LIN {X 35.400,Y 125.914,Z 53.000,A 180.000,B 0.000,C 180.000} C_DIS
LIN {X 35.221,Y 125.886,Z 53.000,A 180.000,B 0.000,C 180.000} C_DIS
LIN {X 35.056,Y 125.857,Z 53.000,A 180.000,B 0.000,C 180.000} C_DIS
LIN {X 34.685,Y 125.774,Z 53.000,A 180.000,B 0.000,C 180.000} C_DIS
LIN {X 34.506,Y 125.726,Z 53.000,A 180.000,B 0.000,C 180.000} C_DIS
LIN {X 34.327,Y 125.674,Z 53.000,A 180.000,B 0.000,C 180.000} C_DIS
LIN {X 34.148,Y 125.619,Z 53.000,A 180.000,B 0.000,C 180.000} C_DIS
LIN {X 33.791,Y 125.491,Z 53.000,A 180.000,B 0.000,C 180.000} C_DIS
LIN {X 33.612,Y 125.417,Z 53.000,A 180.000,B 0.000,C 180.000} C_DIS
LIN {X 33.390,Y 125.321,Z 53.000,A 180.000,B 0.000,C 180.000} C_DIS
LIN {X 33.254,Y 125.258,Z 53.000,A 180.000,B 0.000,C 180.000} C_DIS
LIN {X 32.897,Y 125.076,Z 53.000,A 180.000,B 0.000,C 180.000} C_DIS
LIN {X 32.718,Y 124.971,Z 53.000,A 180.000,B 0.000,C 180.000} C_DIS
LIN {X 32.539,Y 124.865,Z 53.000,A 180.000,B 0.000,C 180.000} C_DIS
LIN {X 32.413,Y 124.785,Z 53.000,A 180.000,B 0.000,C 180.000} C_DIS
LIN {X 32.150,Y 124.606,Z 53.000,A 180.000,B 0.000,C 180.000} C_DIS
LIN {X 32.003,Y 124.497,Z 53.000,A 180.000,B 0.000,C 180.000} C_DIS
LIN {X 31.824,Y 124.359,Z 53.000,A 180.000,B 0.000,C 180.000} C_DIS
LIN {X 31.687,Y 124.248,Z 53.000,A 180.000,B 0.000,C 180.000} C_DIS
LIN {X 31.467,Y 124.055,Z 53.000,A 180.000,B 0.000,C 180.000} C_DIS
LIN {X 31.291,Y 123.891,Z 53.000,A 180.000,B 0.000,C 180.000} C_DIS
LIN {X 31.109,Y 123.709,Z 53.000,A 180.000,B 0.000,C 180.000} C_DIS
LIN {X 30.945,Y 123.533,Z 53.000,A 180.000,B 0.000,C 180.000} C_DIS
LIN {X 30.752,Y 123.313,Z 53.000,A 180.000,B 0.000,C 180.000} C_DIS
LIN {X 30.641,Y 123.176,Z 53.000,A 180.000,B 0.000,C 180.000} C_DIS
LIN {X 30.503,Y 122.997,Z 53.000,A 180.000,B 0.000,C 180.000} C_DIS
LIN {X 30.394,Y 122.850,Z 53.000,A 180.000,B 0.000,C 180.000} C_DIS
LIN {X 30.215,Y 122.587,Z 53.000,A 180.000,B 0.000,C 180.000} C_DIS
LIN {X 30.135,Y 122.461,Z 53.000,A 180.000,B 0.000,C 180.000} C_DIS
LIN {X 30.029,Y 122.282,Z 53.000,A 180.000,B 0.000,C 180.000} C_DIS
LIN {X 29.924,Y 122.103,Z 53.000,A 180.000,B 0.000,C 180.000} C_DIS
LIN {X 29.742,Y 121.746,Z 53.000,A 180.000,B 0.000,C 180.000} C_DIS
LIN {X 29.679,Y 121.610,Z 53.000,A 180.000,B 0.000,C 180.000} C_DIS
LIN {X 29.583,Y 121.388,Z 53.000,A 180.000,B 0.000,C 180.000} C_DIS
LIN {X 29.509,Y 121.209,Z 53.000,A 180.000,B 0.000,C 180.000} C_DIS
LIN {X 29.381,Y 120.852,Z 53.000,A 180.000,B 0.000,C 180.000} C_DIS
LIN {X 29.326,Y 120.673,Z 53.000,A 180.000,B 0.000,C 180.000} C_DIS
LIN {X 29.274,Y 120.494,Z 53.000,A 180.000,B 0.000,C 180.000} C_DIS
LIN {X 29.226,Y 120.315,Z 53.000,A 180.000,B 0.000,C 180.000} C_DIS
LIN {X 29.143,Y 119.944,Z 53.000,A 180.000,B 0.000,C 180.000} C_DIS
LIN {X 29.114,Y 119.779,Z 53.000,A 180.000,B 0.000,C 180.000} C_DIS
LIN {X 29.086,Y 119.600,Z 53.000,A 180.000,B 0.000,C 180.000} C_DIS
LIN {X 29.059,Y 119.422,Z 53.000,A 180.000,B 0.000,C 180.000} C_DIS
LIN {X 29.025,Y 119.064,Z 53.000,A 180.000,B 0.000,C 180.000} C_DIS
LIN {X 29.013,Y 118.885,Z 53.000,A 180.000,B 0.000,C 180.000} C_DIS
LIN {X 29.002,Y 118.528,Z 53.000,A 180.000,B 0.000,C 180.000} C_DIS
LIN {X 29.006,Y 118.349,Z 53.000,A 180.000,B 0.000,C 180.000} C_DIS
LIN {X 29.012,Y 118.170,Z 53.000,A 180.000,B 0.000,C 180.000} C_DIS
LIN {X 29.020,Y 117.991,Z 53.000,A 180.000,B 0.000,C 180.000} C_DIS
LIN {X 29.053,Y 117.634,Z 53.000,A 180.000,B 0.000,C 180.000} C_DIS
LIN {X 29.077,Y 117.455,Z 53.000,A 180.000,B 0.000,C 180.000} C_DIS
LIN {X 29.134,Y 117.098,Z 53.000,A 180.000,B 0.000,C 180.000} C_DIS
LIN {X 29.143,Y 117.056,Z 53.000,A 180.000,B 0.000,C 180.000} C_DIS
LIN {X 29.213,Y 116.740,Z 53.000,A 180.000,B 0.000,C 180.000} C_DIS
LIN {X 29.258,Y 116.561,Z 53.000,A 180.000,B 0.000,C 180.000} C_DIS
LIN {X 29.362,Y 116.204,Z 53.000,A 180.000,B 0.000,C 180.000} C_DIS
LIN {X 29.425,Y 116.025,Z 53.000,A 180.000,B 0.000,C 180.000} C_DIS
LIN {X 29.500,Y 115.816,Z 53.000,A 180.000,B 0.000,C 180.000} C_DIS
LIN {X 29.559,Y 115.667,Z 53.000,A 180.000,B 0.000,C 180.000} C_DIS
LIN {X 29.714,Y 115.310,Z 53.000,A 180.000,B 0.000,C 180.000} C_DIS
LIN {X 29.805,Y 115.131,Z 53.000,A 180.000,B 0.000,C 180.000} C_DIS
LIN {X 29.896,Y 114.952,Z 53.000,A 180.000,B 0.000,C 180.000} C_DIS
LIN {X 29.996,Y 114.774,Z 53.000,A 180.000,B 0.000,C 180.000} C_DIS
LIN {X 30.102,Y 114.595,Z 53.000,A 180.000,B 0.000,C 180.000} C_DIS
LIN {X 30.213,Y 114.416,Z 53.000,A 180.000,B 0.000,C 180.000} C_DIS
LIN {X 30.394,Y 114.150,Z 53.000,A 180.000,B 0.000,C 180.000} C_DIS
LIN {X 30.460,Y 114.058,Z 53.000,A 180.000,B 0.000,C 180.000} C_DIS
LIN {X 30.598,Y 113.880,Z 53.000,A 180.000,B 0.000,C 180.000} C_DIS
LIN {X 30.739,Y 113.701,Z 53.000,A 180.000,B 0.000,C 180.000} C_DIS
LIN {X 30.930,Y 113.484,Z 53.000,A 180.000,B 0.000,C 180.000} C_DIS
LIN {X 31.057,Y 113.343,Z 53.000,A 180.000,B 0.000,C 180.000} C_DIS
LIN {X 31.288,Y 113.112,Z 53.000,A 180.000,B 0.000,C 180.000} C_DIS
LIN {X 31.421,Y 112.986,Z 53.000,A 180.000,B 0.000,C 180.000} C_DIS
LIN {X 31.646,Y 112.788,Z 53.000,A 180.000,B 0.000,C 180.000} C_DIS
LIN {X 31.824,Y 112.641,Z 53.000,A 180.000,B 0.000,C 180.000} C_DIS
LIN {X 32.072,Y 112.450,Z 53.000,A 180.000,B 0.000,C 180.000} C_DIS
LIN {X 32.182,Y 112.373,Z 53.000,A 180.000,B 0.000,C 180.000} C_DIS
LIN {X 32.361,Y 112.251,Z 53.000,A 180.000,B 0.000,C 180.000} C_DIS
LIN {X 32.539,Y 112.135,Z 53.000,A 180.000,B 0.000,C 180.000} C_DIS
LIN {X 32.718,Y 112.029,Z 53.000,A 180.000,B 0.000,C 180.000} C_DIS
LIN {X 32.897,Y 111.924,Z 53.000,A 180.000,B 0.000,C 180.000} C_DIS
LIN {X 33.269,Y 111.734,Z 53.000,A 180.000,B 0.000,C 180.000} C_DIS
LIN {X 33.433,Y 111.660,Z 53.000,A 180.000,B 0.000,C 180.000} C_DIS
LIN {X 33.675,Y 111.556,Z 53.000,A 180.000,B 0.000,C 180.000} C_DIS
LIN {X 33.791,Y 111.509,Z 53.000,A 180.000,B 0.000,C 180.000} C_DIS
LIN {X 34.159,Y 111.377,Z 53.000,A 180.000,B 0.000,C 180.000} C_DIS
LIN {X 34.327,Y 111.326,Z 53.000,A 180.000,B 0.000,C 180.000} C_DIS
LIN {X 34.506,Y 111.274,Z 53.000,A 180.000,B 0.000,C 180.000} C_DIS
LIN {X 34.685,Y 111.226,Z 53.000,A 180.000,B 0.000,C 180.000} C_DIS
LIN {X 35.042,Y 111.146,Z 53.000,A 180.000,B 0.000,C 180.000} C_DIS
LIN {X 35.221,Y 111.114,Z 53.000,A 180.000,B 0.000,C 180.000} C_DIS
LIN {X 35.400,Y 111.086,Z 53.000,A 180.000,B 0.000,C 180.000} C_DIS
LIN {X 35.578,Y 111.059,Z 53.000,A 180.000,B 0.000,C 180.000} C_DIS
LIN {X 35.994,Y 111.019,Z 53.000,A 180.000,B 0.000,C 180.000} C_DIS
LIN {X 36.115,Y 111.013,Z 53.000,A 180.000,B 0.000,C 180.000} C_DIS
LIN {X 36.472,Y 111.002,Z 53.000,A 180.000,B 0.000,C 180.000} C_DIS
LIN {X 36.651,Y 111.006,Z 53.000,A 180.000,B 0.000,C 180.000} C_DIS
LIN {X 36.830,Y 111.012,Z 53.000,A 180.000,B 0.000,C 180.000} C_DIS
LIN {X 37.006,Y 111.019,Z 53.000,A 180.000,B 0.000,C 180.000} C_DIS
LIN {X 37.366,Y 111.053,Z 53.000,A 180.000,B 0.000,C 180.000} C_DIS
LIN {X 37.545,Y 111.077,Z 53.000,A 180.000,B 0.000,C 180.000} C_DIS
LIN {X 37.902,Y 111.134,Z 53.000,A 180.000,B 0.000,C 180.000} C_DIS
LIN {X 38.081,Y 111.173,Z 53.000,A 180.000,B 0.000,C 180.000} C_DIS
LIN {X 38.260,Y 111.213,Z 53.000,A 180.000,B 0.000,C 180.000} C_DIS
LIN {X 38.439,Y 111.258,Z 53.000,A 180.000,B 0.000,C 180.000} C_DIS
LIN {X 38.796,Y 111.362,Z 53.000,A 180.000,B 0.000,C 180.000} C_DIS
LIN {X 38.841,Y 111.377,Z 53.000,A 180.000,B 0.000,C 180.000} C_DIS
LIN {X 39.154,Y 111.489,Z 53.000,A 180.000,B 0.000,C 180.000} C_DIS
LIN {X 39.325,Y 111.556,Z 53.000,A 180.000,B 0.000,C 180.000} C_DIS
LIN {X 39.690,Y 111.714,Z 53.000,A 180.000,B 0.000,C 180.000} C_DIS
LIN {X 39.731,Y 111.734,Z 53.000,A 180.000,B 0.000,C 180.000} C_DIS
LIN {X 40.082,Y 111.913,Z 53.000,A 180.000,B 0.000,C 180.000} C_DIS
LIN {X 40.226,Y 111.996,Z 53.000,A 180.000,B 0.000,C 180.000} C_DIS
LIN {X 40.405,Y 112.102,Z 53.000,A 180.000,B 0.000,C 180.000} C_DIS
LIN {X 40.584,Y 112.213,Z 53.000,A 180.000,B 0.000,C 180.000} C_DIS
LIN {X 40.763,Y 112.335,Z 53.000,A 180.000,B 0.000,C 180.000} C_DIS
LIN {X 40.928,Y 112.450,Z 53.000,A 180.000,B 0.000,C 180.000} C_DIS
LIN {X 41.159,Y 112.628,Z 53.000,A 180.000,B 0.000,C 180.000} C_DIS
LIN {X 41.299,Y 112.739,Z 53.000,A 180.000,B 0.000,C 180.000} C_DIS
LIN {X 41.579,Y 112.986,Z 53.000,A 180.000,B 0.000,C 180.000} C_DIS
LIN {X 41.657,Y 113.057,Z 53.000,A 180.000,B 0.000,C 180.000} C_DIS
LIN {X 41.943,Y 113.343,Z 53.000,A 180.000,B 0.000,C 180.000} C_DIS
LIN {X 42.014,Y 113.421,Z 53.000,A 180.000,B 0.000,C 180.000} C_DIS
LIN {X 42.261,Y 113.701,Z 53.000,A 180.000,B 0.000,C 180.000} C_DIS
LIN {X 42.372,Y 113.841,Z 53.000,A 180.000,B 0.000,C 180.000} C_DIS
LIN {X 42.550,Y 114.072,Z 53.000,A 180.000,B 0.000,C 180.000} C_DIS
LIN {X 42.665,Y 114.237,Z 53.000,A 180.000,B 0.000,C 180.000} C_DIS
LIN {X 42.787,Y 114.416,Z 53.000,A 180.000,B 0.000,C 180.000} C_DIS
LIN {X 42.898,Y 114.595,Z 53.000,A 180.000,B 0.000,C 180.000} C_DIS
LIN {X 43.004,Y 114.774,Z 53.000,A 180.000,B 0.000,C 180.000} C_DIS
LIN {X 43.087,Y 114.918,Z 53.000,A 180.000,B 0.000,C 180.000} C_DIS
LIN {X 43.266,Y 115.269,Z 53.000,A 180.000,B 0.000,C 180.000} C_DIS
LIN {X 43.286,Y 115.310,Z 53.000,A 180.000,B 0.000,C 180.000} C_DIS
LIN {X 43.444,Y 115.675,Z 53.000,A 180.000,B 0.000,C 180.000} C_DIS
LIN {X 43.511,Y 115.846,Z 53.000,A 180.000,B 0.000,C 180.000} C_DIS
LIN {X 43.623,Y 116.159,Z 53.000,A 180.000,B 0.000,C 180.000} C_DIS
LIN {X 43.638,Y 116.204,Z 53.000,A 180.000,B 0.000,C 180.000} C_DIS
LIN {X 43.742,Y 116.561,Z 53.000,A 180.000,B 0.000,C 180.000} C_DIS
LIN {X 43.787,Y 116.740,Z 53.000,A 180.000,B 0.000,C 180.000} C_DIS
LIN {X 43.827,Y 116.919,Z 53.000,A 180.000,B 0.000,C 180.000} C_DIS
LIN {X 43.866,Y 117.098,Z 53.000,A 180.000,B 0.000,C 180.000} C_DIS
LIN {X 43.923,Y 117.455,Z 53.000,A 180.000,B 0.000,C 180.000} C_DIS
LIN {X 43.947,Y 117.634,Z 53.000,A 180.000,B 0.000,C 180.000} C_DIS
LIN {X 43.981,Y 117.994,Z 53.000,A 180.000,B 0.000,C 180.000} C_DIS
LIN {X 43.988,Y 118.170,Z 53.000,A 180.000,B 0.000,C 180.000} C_DIS
LIN {X 43.994,Y 118.349,Z 53.000,A 180.000,B 0.000,C 180.000} C_DIS
LIN {X 43.998,Y 118.528,Z 53.000,A 180.000,B 0.000,C 180.000} C_DIS
LIN {X 43.987,Y 118.885,Z 53.000,A 180.000,B 0.000,C 180.000} C_DIS
LIN {X 43.981,Y 119.006,Z 53.000,A 180.000,B 0.000,C 180.000} C_DIS
LIN {X 43.941,Y 119.422,Z 53.000,A 180.000,B 0.000,C 180.000} C_DIS
LIN {X 43.914,Y 119.600,Z 53.000,A 180.000,B 0.000,C 180.000} C_DIS
LIN {X 43.886,Y 119.779,Z 53.000,A 180.000,B 0.000,C 180.000} C_DIS
LIN {X 43.854,Y 119.958,Z 53.000,A 180.000,B 0.000,C 180.000} C_DIS
LIN {X 43.774,Y 120.315,Z 53.000,A 180.000,B 0.000,C 180.000} C_DIS
LIN {X 43.726,Y 120.494,Z 53.000,A 180.000,B 0.000,C 180.000} C_DIS
LIN {X 43.674,Y 120.673,Z 53.000,A 180.000,B 0.000,C 180.000} C_DIS
LIN {X 43.623,Y 120.841,Z 53.000,A 180.000,B 0.000,C 180.000} C_DIS
LIN {X 43.491,Y 121.209,Z 53.000,A 180.000,B 0.000,C 180.000} C_DIS
LIN {X 43.444,Y 121.325,Z 53.000,A 180.000,B 0.000,C 180.000} C_DIS
LIN {X 43.340,Y 121.567,Z 53.000,A 180.000,B 0.000,C 180.000} C_DIS
LIN {X 43.266,Y 121.731,Z 53.000,A 180.000,B 0.000,C 180.000} C_DIS
LIN {X 43.076,Y 122.103,Z 53.000,A 180.000,B 0.000,C 180.000} C_DIS
LIN {X 42.971,Y 122.282,Z 53.000,A 180.000,B 0.000,C 180.000} C_DIS
LIN {X 42.865,Y 122.461,Z 53.000,A 180.000,B 0.000,C 180.000} C_DIS
LIN {X 42.749,Y 122.639,Z 53.000,A 180.000,B 0.000,C 180.000} C_DIS
LIN {X 42.627,Y 122.818,Z 53.000,A 180.000,B 0.000,C 180.000} C_DIS
LIN {X 42.550,Y 122.928,Z 53.000,A 180.000,B 0.000,C 180.000} C_DIS
LIN {X 42.359,Y 123.176,Z 53.000,A 180.000,B 0.000,C 180.000} C_DIS
LIN {X 42.212,Y 123.354,Z 53.000,A 180.000,B 0.000,C 180.000} C_DIS
LIN {X 42.014,Y 123.579,Z 53.000,A 180.000,B 0.000,C 180.000} C_DIS
LIN {X 41.888,Y 123.712,Z 53.000,A 180.000,B 0.000,C 180.000} C_DIS
LIN {X 41.870,Y 123.729,Z 53.000,A 180.000,B 0.000,C 180.000} C_DIS
; Link Move Starts
LIN {X 41.648,Y 123.952,Z 53.000,A 180.000,B 0.000,C 180.000} C_DIS
LIN {X 41.412,Y 124.161,Z 52.999,A 180.000,B 0.000,C 180.000} C_DIS
LIN {X 41.170,Y 124.363,Z 52.998,A 180.000,B 0.000,C 180.000} C_DIS
LIN {X 40.921,Y 124.556,Z 52.996,A 180.000,B 0.000,C 180.000} C_DIS
LIN {X 40.661,Y 124.734,Z 52.994,A 180.000,B 0.000,C 180.000} C_DIS
LIN {X 40.396,Y 124.904,Z 52.991,A 180.000,B 0.000,C 180.000} C_DIS
LIN {X 40.125,Y 125.064,Z 52.988,A 180.000,B 0.000,C 180.000} C_DIS
LIN {X 39.845,Y 125.208,Z 52.985,A 180.000,B 0.000,C 180.000} C_DIS
LIN {X 39.560,Y 125.343,Z 52.981,A 180.000,B 0.000,C 180.000} C_DIS
LIN {X 39.271,Y 125.468,Z 52.977,A 180.000,B 0.000,C 180.000} C_DIS
LIN {X 38.975,Y 125.575,Z 52.972,A 180.000,B 0.000,C 180.000} C_DIS
LIN {X 38.827,Y 125.628,Z 52.969,A 180.000,B 0.000,C 180.000} C_DIS
LIN {X 38.676,Y 125.673,Z 52.967,A 180.000,B 0.000,C 180.000} C_DIS
LIN {X 38.524,Y 125.717,Z 52.964,A 180.000,B 0.000,C 180.000} C_DIS
LIN {X 38.373,Y 125.761,Z 52.961,A 180.000,B 0.000,C 180.000} C_DIS
LIN {X 38.219,Y 125.796,Z 52.959,A 180.000,B 0.000,C 180.000} C_DIS
LIN {X 38.066,Y 125.830,Z 52.956,A 180.000,B 0.000,C 180.000} C_DIS
LIN {X 37.912,Y 125.864,Z 52.952,A 180.000,B 0.000,C 180.000} C_DIS
LIN {X 37.756,Y 125.889,Z 52.949,A 180.000,B 0.000,C 180.000} C_DIS
LIN {X 37.601,Y 125.914,Z 52.946,A 180.000,B 0.000,C 180.000} C_DIS
LIN {X 37.445,Y 125.939,Z 52.943,A 180.000,B 0.000,C 180.000} C_DIS
LIN {X 37.289,Y 125.954,Z 52.939,A 180.000,B 0.000,C 180.000} C_DIS
LIN {X 37.132,Y 125.969,Z 52.936,A 180.000,B 0.000,C 180.000} C_DIS
LIN {X 36.975,Y 125.984,Z 52.932,A 180.000,B 0.000,C 180.000} C_DIS
LIN {X 36.817,Y 125.989,Z 52.928,A 180.000,B 0.000,C 180.000} C_DIS
LIN {X 36.660,Y 125.994,Z 52.925,A 180.000,B 0.000,C 180.000} C_DIS
LIN {X 36.503,Y 125.999,Z 52.921,A 180.000,B 0.000,C 180.000} C_DIS
LIN {X 36.345,Y 125.994,Z 52.917,A 180.000,B 0.000,C 180.000} C_DIS
LIN {X 36.188,Y 125.989,Z 52.913,A 180.000,B 0.000,C 180.000} C_DIS
LIN {X 36.030,Y 125.984,Z 52.909,A 180.000,B 0.000,C 180.000} C_DIS
LIN {X 35.873,Y 125.969,Z 52.905,A 180.000,B 0.000,C 180.000} C_DIS
LIN {X 35.717,Y 125.954,Z 52.900,A 180.000,B 0.000,C 180.000} C_DIS
LIN {X 35.560,Y 125.940,Z 52.896,A 180.000,B 0.000,C 180.000} C_DIS
LIN {X 35.404,Y 125.915,Z 52.892,A 180.000,B 0.000,C 180.000} C_DIS
LIN {X 35.249,Y 125.890,Z 52.887,A 180.000,B 0.000,C 180.000} C_DIS
LIN {X 35.093,Y 125.866,Z 52.883,A 180.000,B 0.000,C 180.000} C_DIS
LIN {X 34.939,Y 125.831,Z 52.878,A 180.000,B 0.000,C 180.000} C_DIS
LIN {X 34.786,Y 125.797,Z 52.873,A 180.000,B 0.000,C 180.000} C_DIS
LIN {X 34.632,Y 125.762,Z 52.869,A 180.000,B 0.000,C 180.000} C_DIS
LIN {X 34.481,Y 125.718,Z 52.864,A 180.000,B 0.000,C 180.000} C_DIS
LIN {X 34.329,Y 125.674,Z 52.859,A 180.000,B 0.000,C 180.000} C_DIS
LIN {X 34.178,Y 125.630,Z 52.854,A 180.000,B 0.000,C 180.000} C_DIS
LIN {X 34.104,Y 125.603,Z 52.851,A 180.000,B 0.000,C 180.000} C_DIS
LIN {X 34.030,Y 125.577,Z 52.849,A 180.000,B 0.000,C 180.000} C_DIS
LIN {X 33.956,Y 125.550,Z 52.846,A 180.000,B 0.000,C 180.000} C_DIS
LIN {X 33.882,Y 125.523,Z 52.844,A 180.000,B 0.000,C 180.000} C_DIS
LIN {X 33.808,Y 125.497,Z 52.841,A 180.000,B 0.000,C 180.000} C_DIS
LIN {X 33.734,Y 125.470,Z 52.839,A 180.000,B 0.000,C 180.000} C_DIS
LIN {X 33.661,Y 125.438,Z 52.836,A 180.000,B 0.000,C 180.000} C_DIS
LIN {X 33.517,Y 125.376,Z 52.831,A 180.000,B 0.000,C 180.000} C_DIS
LIN {X 33.372,Y 125.313,Z 52.825,A 180.000,B 0.000,C 180.000} C_DIS
LIN {X 33.300,Y 125.282,Z 52.823,A 180.000,B 0.000,C 180.000} C_DIS
LIN {X 33.160,Y 125.210,Z 52.817,A 180.000,B 0.000,C 180.000} C_DIS
LIN {X 33.020,Y 125.139,Z 52.812,A 180.000,B 0.000,C 180.000} C_DIS
LIN {X 32.949,Y 125.103,Z 52.809,A 180.000,B 0.000,C 180.000} C_DIS
LIN {X 32.880,Y 125.067,Z 52.806,A 180.000,B 0.000,C 180.000} C_DIS
LIN {X 32.744,Y 124.986,Z 52.801,A 180.000,B 0.000,C 180.000} C_DIS
LIN {X 32.541,Y 124.866,Z 52.793,A 180.000,B 0.000,C 180.000} C_DIS
LIN {X 32.473,Y 124.825,Z 52.790,A 180.000,B 0.000,C 180.000} C_DIS
LIN {X 32.278,Y 124.693,Z 52.782,A 180.000,B 0.000,C 180.000} C_DIS
LIN {X 32.147,Y 124.604,Z 52.776,A 180.000,B 0.000,C 180.000} C_DIS
LIN {X 32.083,Y 124.559,Z 52.774,A 180.000,B 0.000,C 180.000} C_DIS
LIN {X 31.958,Y 124.463,Z 52.768,A 180.000,B 0.000,C 180.000} C_DIS
LIN {X 31.772,Y 124.318,Z 52.760,A 180.000,B 0.000,C 180.000} C_DIS
LIN {X 31.710,Y 124.269,Z 52.757,A 180.000,B 0.000,C 180.000} C_DIS
LIN {X 31.533,Y 124.113,Z 52.749,A 180.000,B 0.000,C 180.000} C_DIS
LIN {X 31.414,Y 124.008,Z 52.743,A 180.000,B 0.000,C 180.000} C_DIS
LIN {X 31.356,Y 123.956,Z 52.741,A 180.000,B 0.000,C 180.000} C_DIS
LIN {X 31.245,Y 123.844,Z 52.735,A 180.000,B 0.000,C 180.000} C_DIS
LIN {X 31.078,Y 123.677,Z 52.727,A 180.000,B 0.000,C 180.000} C_DIS
LIN {X 31.023,Y 123.621,Z 52.724,A 180.000,B 0.000,C 180.000} C_DIS
LIN {X 30.762,Y 123.325,Z 52.710,A 180.000,B 0.000,C 180.000} C_DIS
LIN {X 30.711,Y 123.265,Z 52.708,A 180.000,B 0.000,C 180.000} C_DIS
LIN {X 30.614,Y 123.141,Z 52.702,A 180.000,B 0.000,C 180.000} C_DIS
LIN {X 30.470,Y 122.954,Z 52.694,A 180.000,B 0.000,C 180.000} C_DIS
LIN {X 30.422,Y 122.891,Z 52.691,A 180.000,B 0.000,C 180.000} C_DIS
LIN {X 30.201,Y 122.566,Z 52.677,A 180.000,B 0.000,C 180.000} C_DIS
LIN {X 30.158,Y 122.500,Z 52.675,A 180.000,B 0.000,C 180.000} C_DIS
LIN {X 30.078,Y 122.364,Z 52.669,A 180.000,B 0.000,C 180.000} C_DIS
LIN {X 29.957,Y 122.161,Z 52.661,A 180.000,B 0.000,C 180.000} C_DIS
LIN {X 29.918,Y 122.092,Z 52.658,A 180.000,B 0.000,C 180.000} C_DIS
LIN {X 29.740,Y 121.742,Z 52.644,A 180.000,B 0.000,C 180.000} C_DIS
LIN {X 29.705,Y 121.671,Z 52.642,A 180.000,B 0.000,C 180.000} C_DIS
LIN {X 29.612,Y 121.454,Z 52.633,A 180.000,B 0.000,C 180.000} C_DIS
LIN {X 29.549,Y 121.309,Z 52.628,A 180.000,B 0.000,C 180.000} C_DIS
LIN {X 29.519,Y 121.236,Z 52.625,A 180.000,B 0.000,C 180.000} C_DIS
LIN {X 29.386,Y 120.866,Z 52.611,A 180.000,B 0.000,C 180.000} C_DIS
LIN {X 29.361,Y 120.791,Z 52.609,A 180.000,B 0.000,C 180.000} C_DIS
LIN {X 29.295,Y 120.564,Z 52.600,A 180.000,B 0.000,C 180.000} C_DIS
LIN {X 29.251,Y 120.413,Z 52.595,A 180.000,B 0.000,C 180.000} C_DIS
LIN {X 29.231,Y 120.337,Z 52.592,A 180.000,B 0.000,C 180.000} C_DIS
LIN {X 29.145,Y 119.953,Z 52.578,A 180.000,B 0.000,C 180.000} C_DIS
LIN {X 29.129,Y 119.875,Z 52.576,A 180.000,B 0.000,C 180.000} C_DIS
LIN {X 29.068,Y 119.487,Z 52.562,A 180.000,B 0.000,C 180.000} C_DIS
LIN {X 29.057,Y 119.408,Z 52.559,A 180.000,B 0.000,C 180.000} C_DIS
LIN {X 29.020,Y 119.016,Z 52.545,A 180.000,B 0.000,C 180.000} C_DIS
LIN {X 29.015,Y 118.938,Z 52.543,A 180.000,B 0.000,C 180.000} C_DIS
LIN {X 29.003,Y 118.544,Z 52.529,A 180.000,B 0.000,C 180.000} C_DIS
LIN {X 29.002,Y 118.466,Z 52.526,A 180.000,B 0.000,C 180.000} C_DIS
LIN {X 29.015,Y 118.072,Z 52.512,A 180.000,B 0.000,C 180.000} C_DIS
LIN {X 29.019,Y 117.993,Z 52.510,A 180.000,B 0.000,C 180.000} C_DIS
LIN {X 29.056,Y 117.601,Z 52.496,A 180.000,B 0.000,C 180.000} C_DIS
LIN {X 29.066,Y 117.523,Z 52.493,A 180.000,B 0.000,C 180.000} C_DIS
LIN {X 29.128,Y 117.134,Z 52.479,A 180.000,B 0.000,C 180.000} C_DIS
LIN {X 29.143,Y 117.057,Z 52.477,A 180.000,B 0.000,C 180.000} C_DIS
LIN {X 29.228,Y 116.673,Z 52.463,A 180.000,B 0.000,C 180.000} C_DIS
LIN {X 29.248,Y 116.596,Z 52.460,A 180.000,B 0.000,C 180.000} C_DIS
LIN {X 29.358,Y 116.218,Z 52.446,A 180.000,B 0.000,C 180.000} C_DIS
LIN {X 29.382,Y 116.143,Z 52.444,A 180.000,B 0.000,C 180.000} C_DIS
LIN {X 29.516,Y 115.773,Z 52.430,A 180.000,B 0.000,C 180.000} C_DIS
LIN {X 29.545,Y 115.700,Z 52.427,A 180.000,B 0.000,C 180.000} C_DIS
LIN {X 29.701,Y 115.338,Z 52.413,A 180.000,B 0.000,C 180.000} C_DIS
LIN {X 29.735,Y 115.267,Z 52.411,A 180.000,B 0.000,C 180.000} C_DIS
LIN {X 29.842,Y 115.057,Z 52.402,A 180.000,B 0.000,C 180.000} C_DIS
LIN {X 29.914,Y 114.916,Z 52.397,A 180.000,B 0.000,C 180.000} C_DIS
LIN {X 29.952,Y 114.848,Z 52.394,A 180.000,B 0.000,C 180.000} C_DIS
LIN {X 30.153,Y 114.509,Z 52.380,A 180.000,B 0.000,C 180.000} C_DIS
LIN {X 30.195,Y 114.442,Z 52.378,A 180.000,B 0.000,C 180.000} C_DIS
LIN {X 30.328,Y 114.247,Z 52.369,A 180.000,B 0.000,C 180.000} C_DIS
LIN {X 30.417,Y 114.117,Z 52.364,A 180.000,B 0.000,C 180.000} C_DIS
LIN {X 30.464,Y 114.053,Z 52.361,A 180.000,B 0.000,C 180.000} C_DIS
LIN {X 30.705,Y 113.742,Z 52.347,A 180.000,B 0.000,C 180.000} C_DIS
LIN {X 30.756,Y 113.682,Z 52.345,A 180.000,B 0.000,C 180.000} C_DIS
LIN {X 30.912,Y 113.505,Z 52.336,A 180.000,B 0.000,C 180.000} C_DIS
LIN {X 31.016,Y 113.387,Z 52.331,A 180.000,B 0.000,C 180.000} C_DIS
LIN {X 31.071,Y 113.330,Z 52.328,A 180.000,B 0.000,C 180.000} C_DIS
LIN {X 31.349,Y 113.051,Z 52.314,A 180.000,B 0.000,C 180.000} C_DIS
LIN {X 31.407,Y 112.998,Z 52.312,A 180.000,B 0.000,C 180.000} C_DIS
LIN {X 31.525,Y 112.894,Z 52.306,A 180.000,B 0.000,C 180.000} C_DIS
LIN {X 31.702,Y 112.738,Z 52.298,A 180.000,B 0.000,C 180.000} C_DIS
LIN {X 31.764,Y 112.688,Z 52.295,A 180.000,B 0.000,C 180.000} C_DIS
LIN {X 31.950,Y 112.543,Z 52.287,A 180.000,B 0.000,C 180.000} C_DIS
LIN {X 32.075,Y 112.447,Z 52.281,A 180.000,B 0.000,C 180.000} C_DIS
LIN {X 32.139,Y 112.402,Z 52.279,A 180.000,B 0.000,C 180.000} C_DIS
LIN {X 32.269,Y 112.313,Z 52.273,A 180.000,B 0.000,C 180.000} C_DIS
LIN {X 32.465,Y 112.180,Z 52.265,A 180.000,B 0.000,C 180.000} C_DIS
LIN {X 32.532,Y 112.139,Z 52.262,A 180.000,B 0.000,C 180.000} C_DIS
LIN {X 32.735,Y 112.019,Z 52.254,A 180.000,B 0.000,C 180.000} C_DIS
LIN {X 32.871,Y 111.939,Z 52.248,A 180.000,B 0.000,C 180.000} C_DIS
LIN {X 32.941,Y 111.902,Z 52.246,A 180.000,B 0.000,C 180.000} C_DIS
LIN {X 33.081,Y 111.830,Z 52.240,A 180.000,B 0.000,C 180.000} C_DIS
LIN {X 33.291,Y 111.723,Z 52.232,A 180.000,B 0.000,C 180.000} C_DIS
LIN {X 33.363,Y 111.691,Z 52.229,A 180.000,B 0.000,C 180.000} C_DIS
LIN {X 33.580,Y 111.597,Z 52.221,A 180.000,B 0.000,C 180.000} C_DIS
LIN {X 33.725,Y 111.534,Z 52.215,A 180.000,B 0.000,C 180.000} C_DIS
LIN {X 33.798,Y 111.507,Z 52.213,A 180.000,B 0.000,C 180.000} C_DIS
LIN {X 33.947,Y 111.453,Z 52.207,A 180.000,B 0.000,C 180.000} C_DIS
LIN {X 34.169,Y 111.373,Z 52.199,A 180.000,B 0.000,C 180.000} C_DIS
LIN {X 34.244,Y 111.350,Z 52.196,A 180.000,B 0.000,C 180.000} C_DIS
LIN {X 34.395,Y 111.306,Z 52.191,A 180.000,B 0.000,C 180.000} C_DIS
LIN {X 34.547,Y 111.263,Z 52.185,A 180.000,B 0.000,C 180.000} C_DIS
LIN {X 34.622,Y 111.241,Z 52.182,A 180.000,B 0.000,C 180.000} C_DIS
LIN {X 34.699,Y 111.223,Z 52.180,A 180.000,B 0.000,C 180.000} C_DIS
LIN {X 34.853,Y 111.188,Z 52.174,A 180.000,B 0.000,C 180.000} C_DIS
LIN {X 35.006,Y 111.154,Z 52.169,A 180.000,B 0.000,C 180.000} C_DIS
LIN {X 35.083,Y 111.137,Z 52.166,A 180.000,B 0.000,C 180.000} C_DIS
LIN {X 35.161,Y 111.124,Z 52.164,A 180.000,B 0.000,C 180.000} C_DIS
LIN {X 35.239,Y 111.111,Z 52.161,A 180.000,B 0.000,C 180.000} C_DIS
LIN {X 35.317,Y 111.099,Z 52.159,A 180.000,B 0.000,C 180.000} C_DIS
LIN {X 35.394,Y 111.087,Z 52.156,A 180.000,B 0.000,C 180.000} C_DIS
LIN {X 35.472,Y 111.074,Z 52.154,A 180.000,B 0.000,C 180.000} C_DIS
LIN {X 35.550,Y 111.062,Z 52.151,A 180.000,B 0.000,C 180.000} C_DIS
LIN {X 35.628,Y 111.054,Z 52.149,A 180.000,B 0.000,C 180.000} C_DIS
LIN {X 35.785,Y 111.039,Z 52.144,A 180.000,B 0.000,C 180.000} C_DIS
LIN {X 35.942,Y 111.024,Z 52.139,A 180.000,B 0.000,C 180.000} C_DIS
LIN {X 36.099,Y 111.014,Z 52.134,A 180.000,B 0.000,C 180.000} C_DIS
LIN {X 36.256,Y 111.009,Z 52.129,A 180.000,B 0.000,C 180.000} C_DIS
LIN {X 36.414,Y 111.004,Z 52.124,A 180.000,B 0.000,C 180.000} C_DIS
LIN {X 36.571,Y 111.003,Z 52.120,A 180.000,B 0.000,C 180.000} C_DIS
LIN {X 36.729,Y 111.008,Z 52.115,A 180.000,B 0.000,C 180.000} C_DIS
LIN {X 36.886,Y 111.013,Z 52.111,A 180.000,B 0.000,C 180.000} C_DIS
LIN {X 37.043,Y 111.023,Z 52.106,A 180.000,B 0.000,C 180.000} C_DIS
LIN {X 37.200,Y 111.038,Z 52.102,A 180.000,B 0.000,C 180.000} C_DIS
LIN {X 37.357,Y 111.053,Z 52.097,A 180.000,B 0.000,C 180.000} C_DIS
LIN {X 37.513,Y 111.072,Z 52.093,A 180.000,B 0.000,C 180.000} C_DIS
LIN {X 37.669,Y 111.097,Z 52.089,A 180.000,B 0.000,C 180.000} C_DIS
LIN {X 37.824,Y 111.121,Z 52.085,A 180.000,B 0.000,C 180.000} C_DIS
LIN {X 37.979,Y 111.151,Z 52.081,A 180.000,B 0.000,C 180.000} C_DIS
LIN {X 38.133,Y 111.185,Z 52.077,A 180.000,B 0.000,C 180.000} C_DIS
LIN {X 38.286,Y 111.219,Z 52.073,A 180.000,B 0.000,C 180.000} C_DIS
LIN {X 38.439,Y 111.258,Z 52.070,A 180.000,B 0.000,C 180.000} C_DIS
LIN {X 38.590,Y 111.302,Z 52.066,A 180.000,B 0.000,C 180.000} C_DIS
LIN {X 38.742,Y 111.346,Z 52.062,A 180.000,B 0.000,C 180.000} C_DIS
LIN {X 38.891,Y 111.395,Z 52.059,A 180.000,B 0.000,C 180.000} C_DIS
LIN {X 39.039,Y 111.448,Z 52.056,A 180.000,B 0.000,C 180.000} C_DIS
LIN {X 39.188,Y 111.502,Z 52.052,A 180.000,B 0.000,C 180.000} C_DIS
LIN {X 39.334,Y 111.560,Z 52.049,A 180.000,B 0.000,C 180.000} C_DIS
LIN {X 39.479,Y 111.622,Z 52.046,A 180.000,B 0.000,C 180.000} C_DIS
LIN {X 39.623,Y 111.685,Z 52.043,A 180.000,B 0.000,C 180.000} C_DIS
LIN {X 39.766,Y 111.752,Z 52.040,A 180.000,B 0.000,C 180.000} C_DIS
LIN {X 39.906,Y 111.823,Z 52.037,A 180.000,B 0.000,C 180.000} C_DIS
LIN {X 40.046,Y 111.895,Z 52.034,A 180.000,B 0.000,C 180.000} C_DIS
LIN {X 40.184,Y 111.971,Z 52.032,A 180.000,B 0.000,C 180.000} C_DIS
LIN {X 40.320,Y 112.051,Z 52.029,A 180.000,B 0.000,C 180.000} C_DIS
LIN {X 40.455,Y 112.131,Z 52.027,A 180.000,B 0.000,C 180.000} C_DIS
LIN {X 40.718,Y 112.305,Z 52.022,A 180.000,B 0.000,C 180.000} C_DIS
LIN {X 40.976,Y 112.486,Z 52.018,A 180.000,B 0.000,C 180.000} C_DIS
LIN {X 41.225,Y 112.679,Z 52.014,A 180.000,B 0.000,C 180.000} C_DIS
LIN {X 41.464,Y 112.884,Z 52.011,A 180.000,B 0.000,C 180.000} C_DIS
LIN {X 41.696,Y 113.097,Z 52.008,A 180.000,B 0.000,C 180.000} C_DIS
LIN {X 41.919,Y 113.319,Z 52.005,A 180.000,B 0.000,C 180.000} C_DIS
LIN {X 42.130,Y 113.553,Z 52.003,A 180.000,B 0.000,C 180.000} C_DIS
LIN {X 42.334,Y 113.793,Z 52.002,A 180.000,B 0.000,C 180.000} C_DIS
LIN {X 42.527,Y 114.042,Z 52.001,A 180.000,B 0.000,C 180.000} C_DIS
LIN {X 42.708,Y 114.300,Z 52.000,A 180.000,B 0.000,C 180.000} C_DIS
LIN {X 42.835,Y 114.494,Z 52.000,A 180.000,B 0.000,C 180.000} C_DIS
; Cutting Move Starts
LIN {X 42.898,Y 114.595,Z 52.000,A 180.000,B 0.000,C 180.000} C_DIS
LIN {X 43.004,Y 114.774,Z 52.000,A 180.000,B 0.000,C 180.000} C_DIS
LIN {X 43.087,Y 114.918,Z 52.000,A 180.000,B 0.000,C 180.000} C_DIS
LIN {X 43.266,Y 115.269,Z 52.000,A 180.000,B 0.000,C 180.000} C_DIS
LIN {X 43.286,Y 115.310,Z 52.000,A 180.000,B 0.000,C 180.000} C_DIS
LIN {X 43.444,Y 115.675,Z 52.000,A 180.000,B 0.000,C 180.000} C_DIS
LIN {X 43.511,Y 115.846,Z 52.000,A 180.000,B 0.000,C 180.000} C_DIS
LIN {X 43.623,Y 116.159,Z 52.000,A 180.000,B 0.000,C 180.000} C_DIS
LIN {X 43.638,Y 116.204,Z 52.000,A 180.000,B 0.000,C 180.000} C_DIS
LIN {X 43.742,Y 116.561,Z 52.000,A 180.000,B 0.000,C 180.000} C_DIS
LIN {X 43.787,Y 116.740,Z 52.000,A 180.000,B 0.000,C 180.000} C_DIS
LIN {X 43.827,Y 116.919,Z 52.000,A 180.000,B 0.000,C 180.000} C_DIS
LIN {X 43.866,Y 117.098,Z 52.000,A 180.000,B 0.000,C 180.000} C_DIS
LIN {X 43.923,Y 117.455,Z 52.000,A 180.000,B 0.000,C 180.000} C_DIS
LIN {X 43.947,Y 117.634,Z 52.000,A 180.000,B 0.000,C 180.000} C_DIS
LIN {X 43.981,Y 117.994,Z 52.000,A 180.000,B 0.000,C 180.000} C_DIS
LIN {X 43.988,Y 118.170,Z 52.000,A 180.000,B 0.000,C 180.000} C_DIS
LIN {X 43.994,Y 118.349,Z 52.000,A 180.000,B 0.000,C 180.000} C_DIS
LIN {X 43.998,Y 118.528,Z 52.000,A 180.000,B 0.000,C 180.000} C_DIS
LIN {X 43.987,Y 118.885,Z 52.000,A 180.000,B 0.000,C 180.000} C_DIS
LIN {X 43.981,Y 119.006,Z 52.000,A 180.000,B 0.000,C 180.000} C_DIS
LIN {X 43.941,Y 119.422,Z 52.000,A 180.000,B 0.000,C 180.000} C_DIS
LIN {X 43.914,Y 119.600,Z 52.000,A 180.000,B 0.000,C 180.000} C_DIS
LIN {X 43.886,Y 119.779,Z 52.000,A 180.000,B 0.000,C 180.000} C_DIS
LIN {X 43.854,Y 119.958,Z 52.000,A 180.000,B 0.000,C 180.000} C_DIS
LIN {X 43.774,Y 120.315,Z 52.000,A 180.000,B 0.000,C 180.000} C_DIS
LIN {X 43.726,Y 120.494,Z 52.000,A 180.000,B 0.000,C 180.000} C_DIS
LIN {X 43.674,Y 120.673,Z 52.000,A 180.000,B 0.000,C 180.000} C_DIS
LIN {X 43.623,Y 120.841,Z 52.000,A 180.000,B 0.000,C 180.000} C_DIS
LIN {X 43.491,Y 121.209,Z 52.000,A 180.000,B 0.000,C 180.000} C_DIS
LIN {X 43.444,Y 121.325,Z 52.000,A 180.000,B 0.000,C 180.000} C_DIS
LIN {X 43.340,Y 121.567,Z 52.000,A 180.000,B 0.000,C 180.000} C_DIS
LIN {X 43.266,Y 121.731,Z 52.000,A 180.000,B 0.000,C 180.000} C_DIS
LIN {X 43.076,Y 122.103,Z 52.000,A 180.000,B 0.000,C 180.000} C_DIS
LIN {X 42.971,Y 122.282,Z 52.000,A 180.000,B 0.000,C 180.000} C_DIS
LIN {X 42.865,Y 122.461,Z 52.000,A 180.000,B 0.000,C 180.000} C_DIS
LIN {X 42.749,Y 122.639,Z 52.000,A 180.000,B 0.000,C 180.000} C_DIS
LIN {X 42.627,Y 122.818,Z 52.000,A 180.000,B 0.000,C 180.000} C_DIS
LIN {X 42.550,Y 122.928,Z 52.000,A 180.000,B 0.000,C 180.000} C_DIS
LIN {X 42.359,Y 123.176,Z 52.000,A 180.000,B 0.000,C 180.000} C_DIS
LIN {X 42.212,Y 123.354,Z 52.000,A 180.000,B 0.000,C 180.000} C_DIS
LIN {X 42.014,Y 123.579,Z 52.000,A 180.000,B 0.000,C 180.000} C_DIS
LIN {X 41.888,Y 123.712,Z 52.000,A 180.000,B 0.000,C 180.000} C_DIS
LIN {X 41.657,Y 123.943,Z 52.000,A 180.000,B 0.000,C 180.000} C_DIS
LIN {X 41.516,Y 124.070,Z 52.000,A 180.000,B 0.000,C 180.000} C_DIS
LIN {X 41.299,Y 124.261,Z 52.000,A 180.000,B 0.000,C 180.000} C_DIS
LIN {X 41.120,Y 124.402,Z 52.000,A 180.000,B 0.000,C 180.000} C_DIS
LIN {X 40.942,Y 124.540,Z 52.000,A 180.000,B 0.000,C 180.000} C_DIS
LIN {X 40.850,Y 124.606,Z 52.000,A 180.000,B 0.000,C 180.000} C_DIS
LIN {X 40.584,Y 124.787,Z 52.000,A 180.000,B 0.000,C 180.000} C_DIS
LIN {X 40.405,Y 124.898,Z 52.000,A 180.000,B 0.000,C 180.000} C_DIS
LIN {X 40.226,Y 125.004,Z 52.000,A 180.000,B 0.000,C 180.000} C_DIS
LIN {X 40.048,Y 125.104,Z 52.000,A 180.000,B 0.000,C 180.000} C_DIS
LIN {X 39.869,Y 125.195,Z 52.000,A 180.000,B 0.000,C 180.000} C_DIS
LIN {X 39.690,Y 125.286,Z 52.000,A 180.000,B 0.000,C 180.000} C_DIS
LIN {X 39.333,Y 125.441,Z 52.000,A 180.000,B 0.000,C 180.000} C_DIS
LIN {X 39.184,Y 125.500,Z 52.000,A 180.000,B 0.000,C 180.000} C_DIS
LIN {X 38.975,Y 125.575,Z 52.000,A 180.000,B 0.000,C 180.000} C_DIS
LIN {X 38.796,Y 125.638,Z 52.000,A 180.000,B 0.000,C 180.000} C_DIS
LIN {X 38.439,Y 125.742,Z 52.000,A 180.000,B 0.000,C 180.000} C_DIS
LIN {X 38.260,Y 125.787,Z 52.000,A 180.000,B 0.000,C 180.000} C_DIS
LIN {X 37.944,Y 125.857,Z 52.000,A 180.000,B 0.000,C 180.000} C_DIS
LIN {X 37.902,Y 125.866,Z 52.000,A 180.000,B 0.000,C 180.000} C_DIS
LIN {X 37.545,Y 125.923,Z 52.000,A 180.000,B 0.000,C 180.000} C_DIS
LIN {X 37.366,Y 125.947,Z 52.000,A 180.000,B 0.000,C 180.000} C_DIS
LIN {X 37.009,Y 125.980,Z 52.000,A 180.000,B 0.000,C 180.000} C_DIS
LIN {X 36.830,Y 125.988,Z 52.000,A 180.000,B 0.000,C 180.000} C_DIS
LIN {X 36.651,Y 125.994,Z 52.000,A 180.000,B 0.000,C 180.000} C_DIS
LIN {X 36.472,Y 125.998,Z 52.000,A 180.000,B 0.000,C 180.000} C_DIS
LIN {X 36.115,Y 125.987,Z 52.000,A 180.000,B 0.000,C 180.000} C_DIS
LIN {X 35.936,Y 125.975,Z 52.000,A 180.000,B 0.000,C 180.000} C_DIS
LIN {X 35.578,Y 125.941,Z 52.000,A 180.000,B 0.000,C 180.000} C_DIS
LIN {X 35.400,Y 125.914,Z 52.000,A 180.000,B 0.000,C 180.000} C_DIS
LIN {X 35.221,Y 125.886,Z 52.000,A 180.000,B 0.000,C 180.000} C_DIS
LIN {X 35.056,Y 125.857,Z 52.000,A 180.000,B 0.000,C 180.000} C_DIS
LIN {X 34.685,Y 125.774,Z 52.000,A 180.000,B 0.000,C 180.000} C_DIS
LIN {X 34.506,Y 125.726,Z 52.000,A 180.000,B 0.000,C 180.000} C_DIS
LIN {X 34.327,Y 125.674,Z 52.000,A 180.000,B 0.000,C 180.000} C_DIS
LIN {X 34.148,Y 125.619,Z 52.000,A 180.000,B 0.000,C 180.000} C_DIS
LIN {X 33.791,Y 125.491,Z 52.000,A 180.000,B 0.000,C 180.000} C_DIS
LIN {X 33.612,Y 125.417,Z 52.000,A 180.000,B 0.000,C 180.000} C_DIS
LIN {X 33.390,Y 125.321,Z 52.000,A 180.000,B 0.000,C 180.000} C_DIS
LIN {X 33.254,Y 125.258,Z 52.000,A 180.000,B 0.000,C 180.000} C_DIS
LIN {X 32.897,Y 125.076,Z 52.000,A 180.000,B 0.000,C 180.000} C_DIS
LIN {X 32.718,Y 124.971,Z 52.000,A 180.000,B 0.000,C 180.000} C_DIS
LIN {X 32.539,Y 124.865,Z 52.000,A 180.000,B 0.000,C 180.000} C_DIS
LIN {X 32.413,Y 124.785,Z 52.000,A 180.000,B 0.000,C 180.000} C_DIS
LIN {X 32.150,Y 124.606,Z 52.000,A 180.000,B 0.000,C 180.000} C_DIS
LIN {X 32.003,Y 124.497,Z 52.000,A 180.000,B 0.000,C 180.000} C_DIS
LIN {X 31.824,Y 124.359,Z 52.000,A 180.000,B 0.000,C 180.000} C_DIS
LIN {X 31.687,Y 124.248,Z 52.000,A 180.000,B 0.000,C 180.000} C_DIS
LIN {X 31.467,Y 124.055,Z 52.000,A 180.000,B 0.000,C 180.000} C_DIS
LIN {X 31.291,Y 123.891,Z 52.000,A 180.000,B 0.000,C 180.000} C_DIS
LIN {X 31.109,Y 123.709,Z 52.000,A 180.000,B 0.000,C 180.000} C_DIS
LIN {X 30.945,Y 123.533,Z 52.000,A 180.000,B 0.000,C 180.000} C_DIS
LIN {X 30.752,Y 123.313,Z 52.000,A 180.000,B 0.000,C 180.000} C_DIS
LIN {X 30.641,Y 123.176,Z 52.000,A 180.000,B 0.000,C 180.000} C_DIS
LIN {X 30.503,Y 122.997,Z 52.000,A 180.000,B 0.000,C 180.000} C_DIS
LIN {X 30.394,Y 122.850,Z 52.000,A 180.000,B 0.000,C 180.000} C_DIS
LIN {X 30.215,Y 122.587,Z 52.000,A 180.000,B 0.000,C 180.000} C_DIS
LIN {X 30.135,Y 122.461,Z 52.000,A 180.000,B 0.000,C 180.000} C_DIS
LIN {X 30.029,Y 122.282,Z 52.000,A 180.000,B 0.000,C 180.000} C_DIS
LIN {X 29.924,Y 122.103,Z 52.000,A 180.000,B 0.000,C 180.000} C_DIS
LIN {X 29.742,Y 121.746,Z 52.000,A 180.000,B 0.000,C 180.000} C_DIS
LIN {X 29.679,Y 121.610,Z 52.000,A 180.000,B 0.000,C 180.000} C_DIS
LIN {X 29.583,Y 121.388,Z 52.000,A 180.000,B 0.000,C 180.000} C_DIS
LIN {X 29.509,Y 121.209,Z 52.000,A 180.000,B 0.000,C 180.000} C_DIS
LIN {X 29.381,Y 120.852,Z 52.000,A 180.000,B 0.000,C 180.000} C_DIS
LIN {X 29.326,Y 120.673,Z 52.000,A 180.000,B 0.000,C 180.000} C_DIS
LIN {X 29.274,Y 120.494,Z 52.000,A 180.000,B 0.000,C 180.000} C_DIS
LIN {X 29.226,Y 120.315,Z 52.000,A 180.000,B 0.000,C 180.000} C_DIS
LIN {X 29.143,Y 119.944,Z 52.000,A 180.000,B 0.000,C 180.000} C_DIS
LIN {X 29.114,Y 119.779,Z 52.000,A 180.000,B 0.000,C 180.000} C_DIS
LIN {X 29.086,Y 119.600,Z 52.000,A 180.000,B 0.000,C 180.000} C_DIS
LIN {X 29.059,Y 119.422,Z 52.000,A 180.000,B 0.000,C 180.000} C_DIS
LIN {X 29.025,Y 119.064,Z 52.000,A 180.000,B 0.000,C 180.000} C_DIS
LIN {X 29.013,Y 118.885,Z 52.000,A 180.000,B 0.000,C 180.000} C_DIS
LIN {X 29.002,Y 118.528,Z 52.000,A 180.000,B 0.000,C 180.000} C_DIS
LIN {X 29.006,Y 118.349,Z 52.000,A 180.000,B 0.000,C 180.000} C_DIS
LIN {X 29.012,Y 118.170,Z 52.000,A 180.000,B 0.000,C 180.000} C_DIS
LIN {X 29.020,Y 117.991,Z 52.000,A 180.000,B 0.000,C 180.000} C_DIS
LIN {X 29.053,Y 117.634,Z 52.000,A 180.000,B 0.000,C 180.000} C_DIS
LIN {X 29.077,Y 117.455,Z 52.000,A 180.000,B 0.000,C 180.000} C_DIS
LIN {X 29.134,Y 117.098,Z 52.000,A 180.000,B 0.000,C 180.000} C_DIS
LIN {X 29.143,Y 117.056,Z 52.000,A 180.000,B 0.000,C 180.000} C_DIS
LIN {X 29.213,Y 116.740,Z 52.000,A 180.000,B 0.000,C 180.000} C_DIS
LIN {X 29.258,Y 116.561,Z 52.000,A 180.000,B 0.000,C 180.000} C_DIS
LIN {X 29.362,Y 116.204,Z 52.000,A 180.000,B 0.000,C 180.000} C_DIS
LIN {X 29.425,Y 116.025,Z 52.000,A 180.000,B 0.000,C 180.000} C_DIS
LIN {X 29.500,Y 115.816,Z 52.000,A 180.000,B 0.000,C 180.000} C_DIS
LIN {X 29.559,Y 115.667,Z 52.000,A 180.000,B 0.000,C 180.000} C_DIS
LIN {X 29.714,Y 115.310,Z 52.000,A 180.000,B 0.000,C 180.000} C_DIS
LIN {X 29.805,Y 115.131,Z 52.000,A 180.000,B 0.000,C 180.000} C_DIS
LIN {X 29.896,Y 114.952,Z 52.000,A 180.000,B 0.000,C 180.000} C_DIS
LIN {X 29.996,Y 114.774,Z 52.000,A 180.000,B 0.000,C 180.000} C_DIS
LIN {X 30.102,Y 114.595,Z 52.000,A 180.000,B 0.000,C 180.000} C_DIS
LIN {X 30.213,Y 114.416,Z 52.000,A 180.000,B 0.000,C 180.000} C_DIS
LIN {X 30.394,Y 114.150,Z 52.000,A 180.000,B 0.000,C 180.000} C_DIS
LIN {X 30.460,Y 114.058,Z 52.000,A 180.000,B 0.000,C 180.000} C_DIS
LIN {X 30.598,Y 113.880,Z 52.000,A 180.000,B 0.000,C 180.000} C_DIS
LIN {X 30.739,Y 113.701,Z 52.000,A 180.000,B 0.000,C 180.000} C_DIS
LIN {X 30.930,Y 113.484,Z 52.000,A 180.000,B 0.000,C 180.000} C_DIS
LIN {X 31.057,Y 113.343,Z 52.000,A 180.000,B 0.000,C 180.000} C_DIS
LIN {X 31.288,Y 113.112,Z 52.000,A 180.000,B 0.000,C 180.000} C_DIS
LIN {X 31.421,Y 112.986,Z 52.000,A 180.000,B 0.000,C 180.000} C_DIS
LIN {X 31.646,Y 112.788,Z 52.000,A 180.000,B 0.000,C 180.000} C_DIS
LIN {X 31.824,Y 112.641,Z 52.000,A 180.000,B 0.000,C 180.000} C_DIS
LIN {X 32.072,Y 112.450,Z 52.000,A 180.000,B 0.000,C 180.000} C_DIS
LIN {X 32.182,Y 112.373,Z 52.000,A 180.000,B 0.000,C 180.000} C_DIS
LIN {X 32.361,Y 112.251,Z 52.000,A 180.000,B 0.000,C 180.000} C_DIS
LIN {X 32.539,Y 112.135,Z 52.000,A 180.000,B 0.000,C 180.000} C_DIS
LIN {X 32.718,Y 112.029,Z 52.000,A 180.000,B 0.000,C 180.000} C_DIS
LIN {X 32.897,Y 111.924,Z 52.000,A 180.000,B 0.000,C 180.000} C_DIS
LIN {X 33.269,Y 111.734,Z 52.000,A 180.000,B 0.000,C 180.000} C_DIS
LIN {X 33.433,Y 111.660,Z 52.000,A 180.000,B 0.000,C 180.000} C_DIS
LIN {X 33.675,Y 111.556,Z 52.000,A 180.000,B 0.000,C 180.000} C_DIS
LIN {X 33.791,Y 111.509,Z 52.000,A 180.000,B 0.000,C 180.000} C_DIS
LIN {X 34.159,Y 111.377,Z 52.000,A 180.000,B 0.000,C 180.000} C_DIS
LIN {X 34.327,Y 111.326,Z 52.000,A 180.000,B 0.000,C 180.000} C_DIS
LIN {X 34.506,Y 111.274,Z 52.000,A 180.000,B 0.000,C 180.000} C_DIS
LIN {X 34.685,Y 111.226,Z 52.000,A 180.000,B 0.000,C 180.000} C_DIS
LIN {X 35.042,Y 111.146,Z 52.000,A 180.000,B 0.000,C 180.000} C_DIS
LIN {X 35.221,Y 111.114,Z 52.000,A 180.000,B 0.000,C 180.000} C_DIS
LIN {X 35.400,Y 111.086,Z 52.000,A 180.000,B 0.000,C 180.000} C_DIS
LIN {X 35.578,Y 111.059,Z 52.000,A 180.000,B 0.000,C 180.000} C_DIS
LIN {X 35.994,Y 111.019,Z 52.000,A 180.000,B 0.000,C 180.000} C_DIS
LIN {X 36.115,Y 111.013,Z 52.000,A 180.000,B 0.000,C 180.000} C_DIS
LIN {X 36.472,Y 111.002,Z 52.000,A 180.000,B 0.000,C 180.000} C_DIS
LIN {X 36.651,Y 111.006,Z 52.000,A 180.000,B 0.000,C 180.000} C_DIS
LIN {X 36.830,Y 111.012,Z 52.000,A 180.000,B 0.000,C 180.000} C_DIS
LIN {X 37.006,Y 111.019,Z 52.000,A 180.000,B 0.000,C 180.000} C_DIS
LIN {X 37.366,Y 111.053,Z 52.000,A 180.000,B 0.000,C 180.000} C_DIS
LIN {X 37.545,Y 111.077,Z 52.000,A 180.000,B 0.000,C 180.000} C_DIS
LIN {X 37.902,Y 111.134,Z 52.000,A 180.000,B 0.000,C 180.000} C_DIS
LIN {X 38.081,Y 111.173,Z 52.000,A 180.000,B 0.000,C 180.000} C_DIS
LIN {X 38.260,Y 111.213,Z 52.000,A 180.000,B 0.000,C 180.000} C_DIS
LIN {X 38.439,Y 111.258,Z 52.000,A 180.000,B 0.000,C 180.000} C_DIS
LIN {X 38.796,Y 111.362,Z 52.000,A 180.000,B 0.000,C 180.000} C_DIS
LIN {X 38.841,Y 111.377,Z 52.000,A 180.000,B 0.000,C 180.000} C_DIS
LIN {X 39.154,Y 111.489,Z 52.000,A 180.000,B 0.000,C 180.000} C_DIS
LIN {X 39.325,Y 111.556,Z 52.000,A 180.000,B 0.000,C 180.000} C_DIS
LIN {X 39.690,Y 111.714,Z 52.000,A 180.000,B 0.000,C 180.000} C_DIS
LIN {X 39.731,Y 111.734,Z 52.000,A 180.000,B 0.000,C 180.000} C_DIS
LIN {X 40.082,Y 111.913,Z 52.000,A 180.000,B 0.000,C 180.000} C_DIS
LIN {X 40.226,Y 111.996,Z 52.000,A 180.000,B 0.000,C 180.000} C_DIS
LIN {X 40.405,Y 112.102,Z 52.000,A 180.000,B 0.000,C 180.000} C_DIS
LIN {X 40.584,Y 112.213,Z 52.000,A 180.000,B 0.000,C 180.000} C_DIS
LIN {X 40.763,Y 112.335,Z 52.000,A 180.000,B 0.000,C 180.000} C_DIS
LIN {X 40.928,Y 112.450,Z 52.000,A 180.000,B 0.000,C 180.000} C_DIS
LIN {X 41.159,Y 112.628,Z 52.000,A 180.000,B 0.000,C 180.000} C_DIS
LIN {X 41.299,Y 112.739,Z 52.000,A 180.000,B 0.000,C 180.000} C_DIS
LIN {X 41.579,Y 112.986,Z 52.000,A 180.000,B 0.000,C 180.000} C_DIS
LIN {X 41.657,Y 113.057,Z 52.000,A 180.000,B 0.000,C 180.000} C_DIS
LIN {X 41.943,Y 113.343,Z 52.000,A 180.000,B 0.000,C 180.000} C_DIS
LIN {X 42.014,Y 113.421,Z 52.000,A 180.000,B 0.000,C 180.000} C_DIS
LIN {X 42.261,Y 113.701,Z 52.000,A 180.000,B 0.000,C 180.000} C_DIS
LIN {X 42.372,Y 113.841,Z 52.000,A 180.000,B 0.000,C 180.000} C_DIS
LIN {X 42.550,Y 114.072,Z 52.000,A 180.000,B 0.000,C 180.000} C_DIS
LIN {X 42.665,Y 114.237,Z 52.000,A 180.000,B 0.000,C 180.000} C_DIS
LIN {X 42.787,Y 114.416,Z 52.000,A 180.000,B 0.000,C 180.000} C_DIS
LIN {X 42.835,Y 114.494,Z 52.000,A 180.000,B 0.000,C 180.000} C_DIS
; Lead Out Move Starts
LIN {X 42.872,Y 114.952,Z 52.000,A 180.000,B 0.000,C 180.000} C_DIS
LIN {X 42.519,Y 115.247,Z 52.000,A 180.000,B 0.000,C 180.000} C_DIS
LIN {X 41.626,Y 115.444,Z 52.000,A 180.000,B 0.000,C 180.000} C_DIS
LIN {X 41.281,Y 115.521,Z 52.146,A 180.000,B 0.000,C 180.000} C_DIS
LIN {X 41.138,Y 115.552,Z 52.500,A 180.000,B 0.000,C 180.000} C_DIS
; Rapid Move Starts
LIN {X 41.138,Y 115.552,Z 95.000,A 180.000,B 0.000,C 180.000} C_DIS
LIN {X 112.331,Y 118.620,Z 95.000,A 180.000,B 0.000,C 180.000} C_DIS
LIN {X 112.331,Y 118.620,Z 58.498,A 180.000,B 0.000,C 180.000} C_DIS
; Plunge Move Starts
$VEL.CP=0.01
LIN {X 112.331,Y 118.620,Z 57.625,A 180.000,B 0.000,C 180.000} C_DIS
; Lead In Move Starts
LIN {X 112.331,Y 118.620,Z 56.500,A 180.000,B 0.000,C 180.000} C_DIS
LIN {X 112.185,Y 118.606,Z 56.146,A 180.000,B 0.000,C 180.000} C_DIS
LIN {X 111.833,Y 118.573,Z 56.000,A 180.000,B 0.000,C 180.000} C_DIS
LIN {X 111.470,Y 118.539,Z 56.000,A 180.000,B 0.000,C 180.000} C_DIS
LIN {X 111.132,Y 118.360,Z 56.000,A 180.000,B 0.000,C 180.000} C_DIS
LIN {X 111.019,Y 117.994,Z 56.000,A 180.000,B 0.000,C 180.000} C_DIS
; Cutting Move Starts
$VEL.CP=0.02
LIN {X 111.053,Y 117.634,Z 56.000,A 180.000,B 0.000,C 180.000} C_DIS
LIN {X 111.077,Y 117.455,Z 56.000,A 180.000,B 0.000,C 180.000} C_DIS
LIN {X 111.134,Y 117.098,Z 56.000,A 180.000,B 0.000,C 180.000} C_DIS
LIN {X 111.173,Y 116.919,Z 56.000,A 180.000,B 0.000,C 180.000} C_DIS
LIN {X 111.213,Y 116.740,Z 56.000,A 180.000,B 0.000,C 180.000} C_DIS
LIN {X 111.258,Y 116.561,Z 56.000,A 180.000,B 0.000,C 180.000} C_DIS
LIN {X 111.362,Y 116.204,Z 56.000,A 180.000,B 0.000,C 180.000} C_DIS
LIN {X 111.377,Y 116.159,Z 56.000,A 180.000,B 0.000,C 180.000} C_DIS
LIN {X 111.489,Y 115.846,Z 56.000,A 180.000,B 0.000,C 180.000} C_DIS
LIN {X 111.556,Y 115.675,Z 56.000,A 180.000,B 0.000,C 180.000} C_DIS
LIN {X 111.714,Y 115.310,Z 56.000,A 180.000,B 0.000,C 180.000} C_DIS
LIN {X 111.734,Y 115.269,Z 56.000,A 180.000,B 0.000,C 180.000} C_DIS
LIN {X 111.913,Y 114.918,Z 56.000,A 180.000,B 0.000,C 180.000} C_DIS
LIN {X 111.996,Y 114.774,Z 56.000,A 180.000,B 0.000,C 180.000} C_DIS
LIN {X 112.102,Y 114.595,Z 56.000,A 180.000,B 0.000,C 180.000} C_DIS
LIN {X 112.213,Y 114.416,Z 56.000,A 180.000,B 0.000,C 180.000} C_DIS
LIN {X 112.335,Y 114.237,Z 56.000,A 180.000,B 0.000,C 180.000} C_DIS
LIN {X 112.450,Y 114.072,Z 56.000,A 180.000,B 0.000,C 180.000} C_DIS
LIN {X 112.628,Y 113.841,Z 56.000,A 180.000,B 0.000,C 180.000} C_DIS
LIN {X 112.739,Y 113.701,Z 56.000,A 180.000,B 0.000,C 180.000} C_DIS
LIN {X 112.986,Y 113.421,Z 56.000,A 180.000,B 0.000,C 180.000} C_DIS
LIN {X 113.057,Y 113.343,Z 56.000,A 180.000,B 0.000,C 180.000} C_DIS
LIN {X 113.343,Y 113.057,Z 56.000,A 180.000,B 0.000,C 180.000} C_DIS
LIN {X 113.421,Y 112.986,Z 56.000,A 180.000,B 0.000,C 180.000} C_DIS
LIN {X 113.701,Y 112.739,Z 56.000,A 180.000,B 0.000,C 180.000} C_DIS
LIN {X 113.841,Y 112.628,Z 56.000,A 180.000,B 0.000,C 180.000} C_DIS
LIN {X 114.072,Y 112.450,Z 56.000,A 180.000,B 0.000,C 180.000} C_DIS
LIN {X 114.237,Y 112.335,Z 56.000,A 180.000,B 0.000,C 180.000} C_DIS
LIN {X 114.416,Y 112.213,Z 56.000,A 180.000,B 0.000,C 180.000} C_DIS
LIN {X 114.595,Y 112.102,Z 56.000,A 180.000,B 0.000,C 180.000} C_DIS
LIN {X 114.774,Y 111.996,Z 56.000,A 180.000,B 0.000,C 180.000} C_DIS
LIN {X 114.918,Y 111.913,Z 56.000,A 180.000,B 0.000,C 180.000} C_DIS
LIN {X 115.269,Y 111.734,Z 56.000,A 180.000,B 0.000,C 180.000} C_DIS
LIN {X 115.310,Y 111.714,Z 56.000,A 180.000,B 0.000,C 180.000} C_DIS
LIN {X 115.675,Y 111.556,Z 56.000,A 180.000,B 0.000,C 180.000} C_DIS
LIN {X 115.846,Y 111.489,Z 56.000,A 180.000,B 0.000,C 180.000} C_DIS
LIN {X 116.159,Y 111.377,Z 56.000,A 180.000,B 0.000,C 180.000} C_DIS
LIN {X 116.204,Y 111.362,Z 56.000,A 180.000,B 0.000,C 180.000} C_DIS
LIN {X 116.561,Y 111.258,Z 56.000,A 180.000,B 0.000,C 180.000} C_DIS
LIN {X 116.740,Y 111.213,Z 56.000,A 180.000,B 0.000,C 180.000} C_DIS
LIN {X 116.919,Y 111.173,Z 56.000,A 180.000,B 0.000,C 180.000} C_DIS
LIN {X 117.098,Y 111.134,Z 56.000,A 180.000,B 0.000,C 180.000} C_DIS
LIN {X 117.455,Y 111.077,Z 56.000,A 180.000,B 0.000,C 180.000} C_DIS
LIN {X 117.634,Y 111.053,Z 56.000,A 180.000,B 0.000,C 180.000} C_DIS
LIN {X 117.994,Y 111.019,Z 56.000,A 180.000,B 0.000,C 180.000} C_DIS
LIN {X 118.170,Y 111.012,Z 56.000,A 180.000,B 0.000,C 180.000} C_DIS
LIN {X 118.349,Y 111.006,Z 56.000,A 180.000,B 0.000,C 180.000} C_DIS
LIN {X 118.528,Y 111.002,Z 56.000,A 180.000,B 0.000,C 180.000} C_DIS
LIN {X 118.885,Y 111.013,Z 56.000,A 180.000,B 0.000,C 180.000} C_DIS
LIN {X 119.006,Y 111.019,Z 56.000,A 180.000,B 0.000,C 180.000} C_DIS
LIN {X 119.422,Y 111.059,Z 56.000,A 180.000,B 0.000,C 180.000} C_DIS
LIN {X 119.600,Y 111.086,Z 56.000,A 180.000,B 0.000,C 180.000} C_DIS
LIN {X 119.779,Y 111.114,Z 56.000,A 180.000,B 0.000,C 180.000} C_DIS
LIN {X 119.958,Y 111.146,Z 56.000,A 180.000,B 0.000,C 180.000} C_DIS
LIN {X 120.315,Y 111.226,Z 56.000,A 180.000,B 0.000,C 180.000} C_DIS
LIN {X 120.494,Y 111.274,Z 56.000,A 180.000,B 0.000,C 180.000} C_DIS
LIN {X 120.673,Y 111.326,Z 56.000,A 180.000,B 0.000,C 180.000} C_DIS
LIN {X 120.841,Y 111.377,Z 56.000,A 180.000,B 0.000,C 180.000} C_DIS
LIN {X 121.209,Y 111.509,Z 56.000,A 180.000,B 0.000,C 180.000} C_DIS
LIN {X 121.325,Y 111.556,Z 56.000,A 180.000,B 0.000,C 180.000} C_DIS
LIN {X 121.567,Y 111.660,Z 56.000,A 180.000,B 0.000,C 180.000} C_DIS
LIN {X 121.731,Y 111.734,Z 56.000,A 180.000,B 0.000,C 180.000} C_DIS
LIN {X 122.103,Y 111.924,Z 56.000,A 180.000,B 0.000,C 180.000} C_DIS
LIN {X 122.282,Y 112.029,Z 56.000,A 180.000,B 0.000,C 180.000} C_DIS
LIN {X 122.461,Y 112.135,Z 56.000,A 180.000,B 0.000,C 180.000} C_DIS
LIN {X 122.639,Y 112.251,Z 56.000,A 180.000,B 0.000,C 180.000} C_DIS
LIN {X 122.818,Y 112.373,Z 56.000,A 180.000,B 0.000,C 180.000} C_DIS
LIN {X 122.928,Y 112.450,Z 56.000,A 180.000,B 0.000,C 180.000} C_DIS
LIN {X 123.176,Y 112.641,Z 56.000,A 180.000,B 0.000,C 180.000} C_DIS
LIN {X 123.354,Y 112.788,Z 56.000,A 180.000,B 0.000,C 180.000} C_DIS
LIN {X 123.579,Y 112.986,Z 56.000,A 180.000,B 0.000,C 180.000} C_DIS
LIN {X 123.712,Y 113.112,Z 56.000,A 180.000,B 0.000,C 180.000} C_DIS
LIN {X 123.943,Y 113.343,Z 56.000,A 180.000,B 0.000,C 180.000} C_DIS
LIN {X 124.070,Y 113.484,Z 56.000,A 180.000,B 0.000,C 180.000} C_DIS
LIN {X 124.261,Y 113.701,Z 56.000,A 180.000,B 0.000,C 180.000} C_DIS
LIN {X 124.402,Y 113.880,Z 56.000,A 180.000,B 0.000,C 180.000} C_DIS
LIN {X 124.540,Y 114.058,Z 56.000,A 180.000,B 0.000,C 180.000} C_DIS
LIN {X 124.606,Y 114.150,Z 56.000,A 180.000,B 0.000,C 180.000} C_DIS
LIN {X 124.787,Y 114.416,Z 56.000,A 180.000,B 0.000,C 180.000} C_DIS
LIN {X 124.898,Y 114.595,Z 56.000,A 180.000,B 0.000,C 180.000} C_DIS
LIN {X 125.004,Y 114.774,Z 56.000,A 180.000,B 0.000,C 180.000} C_DIS
LIN {X 125.104,Y 114.952,Z 56.000,A 180.000,B 0.000,C 180.000} C_DIS
LIN {X 125.195,Y 115.131,Z 56.000,A 180.000,B 0.000,C 180.000} C_DIS
LIN {X 125.286,Y 115.310,Z 56.000,A 180.000,B 0.000,C 180.000} C_DIS
LIN {X 125.441,Y 115.667,Z 56.000,A 180.000,B 0.000,C 180.000} C_DIS
LIN {X 125.500,Y 115.816,Z 56.000,A 180.000,B 0.000,C 180.000} C_DIS
LIN {X 125.575,Y 116.025,Z 56.000,A 180.000,B 0.000,C 180.000} C_DIS
LIN {X 125.638,Y 116.204,Z 56.000,A 180.000,B 0.000,C 180.000} C_DIS
LIN {X 125.742,Y 116.561,Z 56.000,A 180.000,B 0.000,C 180.000} C_DIS
LIN {X 125.787,Y 116.740,Z 56.000,A 180.000,B 0.000,C 180.000} C_DIS
LIN {X 125.857,Y 117.056,Z 56.000,A 180.000,B 0.000,C 180.000} C_DIS
LIN {X 125.866,Y 117.098,Z 56.000,A 180.000,B 0.000,C 180.000} C_DIS
LIN {X 125.923,Y 117.455,Z 56.000,A 180.000,B 0.000,C 180.000} C_DIS
LIN {X 125.947,Y 117.634,Z 56.000,A 180.000,B 0.000,C 180.000} C_DIS
LIN {X 125.980,Y 117.991,Z 56.000,A 180.000,B 0.000,C 180.000} C_DIS
LIN {X 125.988,Y 118.170,Z 56.000,A 180.000,B 0.000,C 180.000} C_DIS
LIN {X 125.994,Y 118.349,Z 56.000,A 180.000,B 0.000,C 180.000} C_DIS
LIN {X 125.998,Y 118.528,Z 56.000,A 180.000,B 0.000,C 180.000} C_DIS
LIN {X 125.987,Y 118.885,Z 56.000,A 180.000,B 0.000,C 180.000} C_DIS
LIN {X 125.975,Y 119.064,Z 56.000,A 180.000,B 0.000,C 180.000} C_DIS
LIN {X 125.941,Y 119.422,Z 56.000,A 180.000,B 0.000,C 180.000} C_DIS
LIN {X 125.914,Y 119.600,Z 56.000,A 180.000,B 0.000,C 180.000} C_DIS
LIN {X 125.886,Y 119.779,Z 56.000,A 180.000,B 0.000,C 180.000} C_DIS
LIN {X 125.857,Y 119.944,Z 56.000,A 180.000,B 0.000,C 180.000} C_DIS
LIN {X 125.774,Y 120.315,Z 56.000,A 180.000,B 0.000,C 180.000} C_DIS
LIN {X 125.726,Y 120.494,Z 56.000,A 180.000,B 0.000,C 180.000} C_DIS
LIN {X 125.674,Y 120.673,Z 56.000,A 180.000,B 0.000,C 180.000} C_DIS
LIN {X 125.619,Y 120.852,Z 56.000,A 180.000,B 0.000,C 180.000} C_DIS
LIN {X 125.491,Y 121.209,Z 56.000,A 180.000,B 0.000,C 180.000} C_DIS
LIN {X 125.417,Y 121.388,Z 56.000,A 180.000,B 0.000,C 180.000} C_DIS
LIN {X 125.321,Y 121.610,Z 56.000,A 180.000,B 0.000,C 180.000} C_DIS
LIN {X 125.258,Y 121.746,Z 56.000,A 180.000,B 0.000,C 180.000} C_DIS
LIN {X 125.076,Y 122.103,Z 56.000,A 180.000,B 0.000,C 180.000} C_DIS
LIN {X 124.971,Y 122.282,Z 56.000,A 180.000,B 0.000,C 180.000} C_DIS
LIN {X 124.865,Y 122.461,Z 56.000,A 180.000,B 0.000,C 180.000} C_DIS
LIN {X 124.785,Y 122.587,Z 56.000,A 180.000,B 0.000,C 180.000} C_DIS
LIN {X 124.606,Y 122.850,Z 56.000,A 180.000,B 0.000,C 180.000} C_DIS
LIN {X 124.497,Y 122.997,Z 56.000,A 180.000,B 0.000,C 180.000} C_DIS
LIN {X 124.359,Y 123.176,Z 56.000,A 180.000,B 0.000,C 180.000} C_DIS
LIN {X 124.248,Y 123.313,Z 56.000,A 180.000,B 0.000,C 180.000} C_DIS
LIN {X 124.055,Y 123.533,Z 56.000,A 180.000,B 0.000,C 180.000} C_DIS
LIN {X 123.891,Y 123.709,Z 56.000,A 180.000,B 0.000,C 180.000} C_DIS
LIN {X 123.709,Y 123.891,Z 56.000,A 180.000,B 0.000,C 180.000} C_DIS
LIN {X 123.533,Y 124.055,Z 56.000,A 180.000,B 0.000,C 180.000} C_DIS
LIN {X 123.313,Y 124.248,Z 56.000,A 180.000,B 0.000,C 180.000} C_DIS
LIN {X 123.176,Y 124.359,Z 56.000,A 180.000,B 0.000,C 180.000} C_DIS
LIN {X 122.997,Y 124.497,Z 56.000,A 180.000,B 0.000,C 180.000} C_DIS
LIN {X 122.850,Y 124.606,Z 56.000,A 180.000,B 0.000,C 180.000} C_DIS
LIN {X 122.587,Y 124.785,Z 56.000,A 180.000,B 0.000,C 180.000} C_DIS
LIN {X 122.461,Y 124.865,Z 56.000,A 180.000,B 0.000,C 180.000} C_DIS
LIN {X 122.282,Y 124.971,Z 56.000,A 180.000,B 0.000,C 180.000} C_DIS
LIN {X 122.103,Y 125.076,Z 56.000,A 180.000,B 0.000,C 180.000} C_DIS
LIN {X 121.746,Y 125.258,Z 56.000,A 180.000,B 0.000,C 180.000} C_DIS
LIN {X 121.610,Y 125.321,Z 56.000,A 180.000,B 0.000,C 180.000} C_DIS
LIN {X 121.388,Y 125.417,Z 56.000,A 180.000,B 0.000,C 180.000} C_DIS
LIN {X 121.209,Y 125.491,Z 56.000,A 180.000,B 0.000,C 180.000} C_DIS
LIN {X 120.852,Y 125.619,Z 56.000,A 180.000,B 0.000,C 180.000} C_DIS
LIN {X 120.673,Y 125.674,Z 56.000,A 180.000,B 0.000,C 180.000} C_DIS
LIN {X 120.494,Y 125.726,Z 56.000,A 180.000,B 0.000,C 180.000} C_DIS
LIN {X 120.315,Y 125.774,Z 56.000,A 180.000,B 0.000,C 180.000} C_DIS
LIN {X 119.944,Y 125.857,Z 56.000,A 180.000,B 0.000,C 180.000} C_DIS
LIN {X 119.779,Y 125.886,Z 56.000,A 180.000,B 0.000,C 180.000} C_DIS
LIN {X 119.600,Y 125.914,Z 56.000,A 180.000,B 0.000,C 180.000} C_DIS
LIN {X 119.422,Y 125.941,Z 56.000,A 180.000,B 0.000,C 180.000} C_DIS
LIN {X 119.064,Y 125.975,Z 56.000,A 180.000,B 0.000,C 180.000} C_DIS
LIN {X 118.885,Y 125.987,Z 56.000,A 180.000,B 0.000,C 180.000} C_DIS
LIN {X 118.528,Y 125.998,Z 56.000,A 180.000,B 0.000,C 180.000} C_DIS
LIN {X 118.349,Y 125.994,Z 56.000,A 180.000,B 0.000,C 180.000} C_DIS
LIN {X 118.170,Y 125.988,Z 56.000,A 180.000,B 0.000,C 180.000} C_DIS
LIN {X 117.991,Y 125.980,Z 56.000,A 180.000,B 0.000,C 180.000} C_DIS
LIN {X 117.634,Y 125.947,Z 56.000,A 180.000,B 0.000,C 180.000} C_DIS
LIN {X 117.455,Y 125.923,Z 56.000,A 180.000,B 0.000,C 180.000} C_DIS
LIN {X 117.098,Y 125.866,Z 56.000,A 180.000,B 0.000,C 180.000} C_DIS
LIN {X 117.056,Y 125.857,Z 56.000,A 180.000,B 0.000,C 180.000} C_DIS
LIN {X 116.740,Y 125.787,Z 56.000,A 180.000,B 0.000,C 180.000} C_DIS
LIN {X 116.561,Y 125.742,Z 56.000,A 180.000,B 0.000,C 180.000} C_DIS
LIN {X 116.204,Y 125.638,Z 56.000,A 180.000,B 0.000,C 180.000} C_DIS
LIN {X 116.025,Y 125.575,Z 56.000,A 180.000,B 0.000,C 180.000} C_DIS
LIN {X 115.816,Y 125.500,Z 56.000,A 180.000,B 0.000,C 180.000} C_DIS
LIN {X 115.667,Y 125.441,Z 56.000,A 180.000,B 0.000,C 180.000} C_DIS
LIN {X 115.310,Y 125.286,Z 56.000,A 180.000,B 0.000,C 180.000} C_DIS
LIN {X 115.131,Y 125.195,Z 56.000,A 180.000,B 0.000,C 180.000} C_DIS
LIN {X 114.952,Y 125.104,Z 56.000,A 180.000,B 0.000,C 180.000} C_DIS
LIN {X 114.774,Y 125.004,Z 56.000,A 180.000,B 0.000,C 180.000} C_DIS
LIN {X 114.595,Y 124.898,Z 56.000,A 180.000,B 0.000,C 180.000} C_DIS
LIN {X 114.416,Y 124.787,Z 56.000,A 180.000,B 0.000,C 180.000} C_DIS
LIN {X 114.150,Y 124.606,Z 56.000,A 180.000,B 0.000,C 180.000} C_DIS
LIN {X 114.058,Y 124.540,Z 56.000,A 180.000,B 0.000,C 180.000} C_DIS
LIN {X 113.880,Y 124.402,Z 56.000,A 180.000,B 0.000,C 180.000} C_DIS
LIN {X 113.701,Y 124.261,Z 56.000,A 180.000,B 0.000,C 180.000} C_DIS
LIN {X 113.484,Y 124.070,Z 56.000,A 180.000,B 0.000,C 180.000} C_DIS
LIN {X 113.343,Y 123.943,Z 56.000,A 180.000,B 0.000,C 180.000} C_DIS
LIN {X 113.112,Y 123.712,Z 56.000,A 180.000,B 0.000,C 180.000} C_DIS
LIN {X 112.986,Y 123.579,Z 56.000,A 180.000,B 0.000,C 180.000} C_DIS
LIN {X 112.788,Y 123.354,Z 56.000,A 180.000,B 0.000,C 180.000} C_DIS
LIN {X 112.641,Y 123.176,Z 56.000,A 180.000,B 0.000,C 180.000} C_DIS
LIN {X 112.450,Y 122.928,Z 56.000,A 180.000,B 0.000,C 180.000} C_DIS
LIN {X 112.373,Y 122.818,Z 56.000,A 180.000,B 0.000,C 180.000} C_DIS
LIN {X 112.251,Y 122.639,Z 56.000,A 180.000,B 0.000,C 180.000} C_DIS
LIN {X 112.135,Y 122.461,Z 56.000,A 180.000,B 0.000,C 180.000} C_DIS
LIN {X 112.029,Y 122.282,Z 56.000,A 180.000,B 0.000,C 180.000} C_DIS
LIN {X 111.924,Y 122.103,Z 56.000,A 180.000,B 0.000,C 180.000} C_DIS
LIN {X 111.734,Y 121.731,Z 56.000,A 180.000,B 0.000,C 180.000} C_DIS
LIN {X 111.660,Y 121.567,Z 56.000,A 180.000,B 0.000,C 180.000} C_DIS
LIN {X 111.556,Y 121.325,Z 56.000,A 180.000,B 0.000,C 180.000} C_DIS
LIN {X 111.509,Y 121.209,Z 56.000,A 180.000,B 0.000,C 180.000} C_DIS
LIN {X 111.377,Y 120.841,Z 56.000,A 180.000,B 0.000,C 180.000} C_DIS
LIN {X 111.326,Y 120.673,Z 56.000,A 180.000,B 0.000,C 180.000} C_DIS
LIN {X 111.274,Y 120.494,Z 56.000,A 180.000,B 0.000,C 180.000} C_DIS
LIN {X 111.226,Y 120.315,Z 56.000,A 180.000,B 0.000,C 180.000} C_DIS
LIN {X 111.146,Y 119.958,Z 56.000,A 180.000,B 0.000,C 180.000} C_DIS
LIN {X 111.114,Y 119.779,Z 56.000,A 180.000,B 0.000,C 180.000} C_DIS
LIN {X 111.086,Y 119.600,Z 56.000,A 180.000,B 0.000,C 180.000} C_DIS
LIN {X 111.059,Y 119.422,Z 56.000,A 180.000,B 0.000,C 180.000} C_DIS
LIN {X 111.019,Y 119.006,Z 56.000,A 180.000,B 0.000,C 180.000} C_DIS
LIN {X 111.013,Y 118.885,Z 56.000,A 180.000,B 0.000,C 180.000} C_DIS
LIN {X 111.002,Y 118.528,Z 56.000,A 180.000,B 0.000,C 180.000} C_DIS
LIN {X 111.006,Y 118.349,Z 56.000,A 180.000,B 0.000,C 180.000} C_DIS
LIN {X 111.012,Y 118.170,Z 56.000,A 180.000,B 0.000,C 180.000} C_DIS
LIN {X 111.019,Y 117.994,Z 56.000,A 180.000,B 0.000,C 180.000} C_DIS
; Link Move Starts
LIN {X 111.049,Y 117.680,Z 56.000,A 180.000,B 0.000,C 180.000} C_DIS
LIN {X 111.091,Y 117.368,Z 55.999,A 180.000,B 0.000,C 180.000} C_DIS
LIN {X 111.142,Y 117.057,Z 55.998,A 180.000,B 0.000,C 180.000} C_DIS
LIN {X 111.211,Y 116.750,Z 55.996,A 180.000,B 0.000,C 180.000} C_DIS
LIN {X 111.292,Y 116.446,Z 55.994,A 180.000,B 0.000,C 180.000} C_DIS
LIN {X 111.382,Y 116.144,Z 55.991,A 180.000,B 0.000,C 180.000} C_DIS
LIN {X 111.489,Y 115.848,Z 55.988,A 180.000,B 0.000,C 180.000} C_DIS
LIN {X 111.607,Y 115.556,Z 55.985,A 180.000,B 0.000,C 180.000} C_DIS
LIN {X 111.735,Y 115.268,Z 55.981,A 180.000,B 0.000,C 180.000} C_DIS
LIN {X 111.878,Y 114.987,Z 55.977,A 180.000,B 0.000,C 180.000} C_DIS
LIN {X 112.032,Y 114.713,Z 55.972,A 180.000,B 0.000,C 180.000} C_DIS
LIN {X 112.112,Y 114.577,Z 55.969,A 180.000,B 0.000,C 180.000} C_DIS
LIN {X 112.195,Y 114.443,Z 55.967,A 180.000,B 0.000,C 180.000} C_DIS
LIN {X 112.284,Y 114.313,Z 55.964,A 180.000,B 0.000,C 180.000} C_DIS
LIN {X 112.372,Y 114.182,Z 55.961,A 180.000,B 0.000,C 180.000} C_DIS
LIN {X 112.463,Y 114.054,Z 55.959,A 180.000,B 0.000,C 180.000} C_DIS
LIN {X 112.560,Y 113.929,Z 55.956,A 180.000,B 0.000,C 180.000} C_DIS
LIN {X 112.656,Y 113.805,Z 55.952,A 180.000,B 0.000,C 180.000} C_DIS
LIN {X 112.755,Y 113.683,Z 55.949,A 180.000,B 0.000,C 180.000} C_DIS
LIN {X 112.859,Y 113.564,Z 55.946,A 180.000,B 0.000,C 180.000} C_DIS
LIN {X 112.964,Y 113.446,Z 55.943,A 180.000,B 0.000,C 180.000} C_DIS
LIN {X 113.070,Y 113.330,Z 55.939,A 180.000,B 0.000,C 180.000} C_DIS
LIN {X 113.181,Y 113.219,Z 55.936,A 180.000,B 0.000,C 180.000} C_DIS
LIN {X 113.293,Y 113.108,Z 55.932,A 180.000,B 0.000,C 180.000} C_DIS
LIN {X 113.407,Y 112.999,Z 55.928,A 180.000,B 0.000,C 180.000} C_DIS
LIN {X 113.525,Y 112.894,Z 55.925,A 180.000,B 0.000,C 180.000} C_DIS
LIN {X 113.643,Y 112.790,Z 55.921,A 180.000,B 0.000,C 180.000} C_DIS
LIN {X 113.763,Y 112.689,Z 55.917,A 180.000,B 0.000,C 180.000} C_DIS
LIN {X 113.888,Y 112.592,Z 55.913,A 180.000,B 0.000,C 180.000} C_DIS
LIN {X 114.012,Y 112.496,Z 55.909,A 180.000,B 0.000,C 180.000} C_DIS
LIN {X 114.139,Y 112.402,Z 55.905,A 180.000,B 0.000,C 180.000} C_DIS
LIN {X 114.269,Y 112.313,Z 55.900,A 180.000,B 0.000,C 180.000} C_DIS
LIN {X 114.399,Y 112.225,Z 55.896,A 180.000,B 0.000,C 180.000} C_DIS
LIN {X 114.531,Y 112.139,Z 55.892,A 180.000,B 0.000,C 180.000} C_DIS
LIN {X 114.667,Y 112.059,Z 55.887,A 180.000,B 0.000,C 180.000} C_DIS
LIN {X 114.803,Y 111.979,Z 55.883,A 180.000,B 0.000,C 180.000} C_DIS
LIN {X 114.940,Y 111.902,Z 55.878,A 180.000,B 0.000,C 180.000} C_DIS
LIN {X 115.080,Y 111.831,Z 55.873,A 180.000,B 0.000,C 180.000} C_DIS
LIN {X 115.221,Y 111.759,Z 55.869,A 180.000,B 0.000,C 180.000} C_DIS
LIN {X 115.363,Y 111.691,Z 55.864,A 180.000,B 0.000,C 180.000} C_DIS
LIN {X 115.507,Y 111.628,Z 55.859,A 180.000,B 0.000,C 180.000} C_DIS
LIN {X 115.652,Y 111.566,Z 55.854,A 180.000,B 0.000,C 180.000} C_DIS
LIN {X 115.724,Y 111.535,Z 55.851,A 180.000,B 0.000,C 180.000} C_DIS
LIN {X 115.798,Y 111.507,Z 55.849,A 180.000,B 0.000,C 180.000} C_DIS
LIN {X 115.872,Y 111.480,Z 55.846,A 180.000,B 0.000,C 180.000} C_DIS
LIN {X 115.946,Y 111.454,Z 55.844,A 180.000,B 0.000,C 180.000} C_DIS
LIN {X 116.020,Y 111.427,Z 55.841,A 180.000,B 0.000,C 180.000} C_DIS
LIN {X 116.168,Y 111.373,Z 55.836,A 180.000,B 0.000,C 180.000} C_DIS
LIN {X 116.244,Y 111.351,Z 55.833,A 180.000,B 0.000,C 180.000} C_DIS
LIN {X 116.395,Y 111.307,Z 55.828,A 180.000,B 0.000,C 180.000} C_DIS
LIN {X 116.546,Y 111.263,Z 55.823,A 180.000,B 0.000,C 180.000} C_DIS
LIN {X 116.622,Y 111.241,Z 55.820,A 180.000,B 0.000,C 180.000} C_DIS
LIN {X 116.698,Y 111.223,Z 55.817,A 180.000,B 0.000,C 180.000} C_DIS
LIN {X 116.852,Y 111.188,Z 55.812,A 180.000,B 0.000,C 180.000} C_DIS
LIN {X 117.083,Y 111.137,Z 55.804,A 180.000,B 0.000,C 180.000} C_DIS
LIN {X 117.160,Y 111.124,Z 55.801,A 180.000,B 0.000,C 180.000} C_DIS
LIN {X 117.394,Y 111.087,Z 55.793,A 180.000,B 0.000,C 180.000} C_DIS
LIN {X 117.549,Y 111.062,Z 55.787,A 180.000,B 0.000,C 180.000} C_DIS
LIN {X 117.628,Y 111.054,Z 55.785,A 180.000,B 0.000,C 180.000} C_DIS
LIN {X 117.784,Y 111.039,Z 55.779,A 180.000,B 0.000,C 180.000} C_DIS
LIN {X 118.020,Y 111.017,Z 55.771,A 180.000,B 0.000,C 180.000} C_DIS
LIN {X 118.098,Y 111.014,Z 55.768,A 180.000,B 0.000,C 180.000} C_DIS
LIN {X 118.334,Y 111.006,Z 55.760,A 180.000,B 0.000,C 180.000} C_DIS
LIN {X 118.492,Y 111.001,Z 55.754,A 180.000,B 0.000,C 180.000} C_DIS
LIN {X 118.571,Y 111.003,Z 55.752,A 180.000,B 0.000,C 180.000} C_DIS
LIN {X 118.728,Y 111.008,Z 55.746,A 180.000,B 0.000,C 180.000} C_DIS
LIN {X 118.964,Y 111.016,Z 55.738,A 180.000,B 0.000,C 180.000} C_DIS
LIN {X 119.043,Y 111.023,Z 55.735,A 180.000,B 0.000,C 180.000} C_DIS
LIN {X 119.278,Y 111.045,Z 55.727,A 180.000,B 0.000,C 180.000} C_DIS
LIN {X 119.435,Y 111.060,Z 55.721,A 180.000,B 0.000,C 180.000} C_DIS
LIN {X 119.513,Y 111.072,Z 55.719,A 180.000,B 0.000,C 180.000} C_DIS
LIN {X 119.668,Y 111.097,Z 55.713,A 180.000,B 0.000,C 180.000} C_DIS
LIN {X 119.901,Y 111.133,Z 55.705,A 180.000,B 0.000,C 180.000} C_DIS
LIN {X 119.978,Y 111.150,Z 55.702,A 180.000,B 0.000,C 180.000} C_DIS
LIN {X 120.363,Y 111.236,Z 55.688,A 180.000,B 0.000,C 180.000} C_DIS
LIN {X 120.438,Y 111.258,Z 55.686,A 180.000,B 0.000,C 180.000} C_DIS
LIN {X 120.590,Y 111.302,Z 55.680,A 180.000,B 0.000,C 180.000} C_DIS
LIN {X 120.817,Y 111.368,Z 55.672,A 180.000,B 0.000,C 180.000} C_DIS
LIN {X 120.891,Y 111.395,Z 55.669,A 180.000,B 0.000,C 180.000} C_DIS
LIN {X 121.187,Y 111.501,Z 55.658,A 180.000,B 0.000,C 180.000} C_DIS
LIN {X 121.261,Y 111.528,Z 55.655,A 180.000,B 0.000,C 180.000} C_DIS
LIN {X 121.406,Y 111.591,Z 55.650,A 180.000,B 0.000,C 180.000} C_DIS
LIN {X 121.623,Y 111.684,Z 55.642,A 180.000,B 0.000,C 180.000} C_DIS
LIN {X 121.695,Y 111.716,Z 55.639,A 180.000,B 0.000,C 180.000} C_DIS
LIN {X 122.046,Y 111.895,Z 55.625,A 180.000,B 0.000,C 180.000} C_DIS
LIN {X 122.116,Y 111.931,Z 55.622,A 180.000,B 0.000,C 180.000} C_DIS
LIN {X 122.319,Y 112.051,Z 55.614,A 180.000,B 0.000,C 180.000} C_DIS
LIN {X 122.455,Y 112.131,Z 55.609,A 180.000,B 0.000,C 180.000} C_DIS
LIN {X 122.522,Y 112.171,Z 55.606,A 180.000,B 0.000,C 180.000} C_DIS
LIN {X 122.848,Y 112.393,Z 55.592,A 180.000,B 0.000,C 180.000} C_DIS
LIN {X 122.913,Y 112.437,Z 55.589,A 180.000,B 0.000,C 180.000} C_DIS
LIN {X 123.224,Y 112.679,Z 55.576,A 180.000,B 0.000,C 180.000} C_DIS
LIN {X 123.286,Y 112.727,Z 55.573,A 180.000,B 0.000,C 180.000} C_DIS
LIN {X 123.581,Y 112.988,Z 55.559,A 180.000,B 0.000,C 180.000} C_DIS
LIN {X 123.640,Y 113.040,Z 55.556,A 180.000,B 0.000,C 180.000} C_DIS
LIN {X 123.918,Y 113.319,Z 55.543,A 180.000,B 0.000,C 180.000} C_DIS
LIN {X 123.974,Y 113.375,Z 55.540,A 180.000,B 0.000,C 180.000} C_DIS
LIN {X 124.234,Y 113.670,Z 55.526,A 180.000,B 0.000,C 180.000} C_DIS
LIN {X 124.286,Y 113.730,Z 55.523,A 180.000,B 0.000,C 180.000} C_DIS
LIN {X 124.527,Y 114.041,Z 55.510,A 180.000,B 0.000,C 180.000} C_DIS
LIN {X 124.575,Y 114.104,Z 55.507,A 180.000,B 0.000,C 180.000} C_DIS
LIN {X 124.796,Y 114.430,Z 55.493,A 180.000,B 0.000,C 180.000} C_DIS
LIN {X 124.839,Y 114.495,Z 55.490,A 180.000,B 0.000,C 180.000} C_DIS
LIN {X 125.040,Y 114.834,Z 55.477,A 180.000,B 0.000,C 180.000} C_DIS
LIN {X 125.079,Y 114.903,Z 55.474,A 180.000,B 0.000,C 180.000} C_DIS
LIN {X 125.258,Y 115.253,Z 55.460,A 180.000,B 0.000,C 180.000} C_DIS
LIN {X 125.292,Y 115.324,Z 55.457,A 180.000,B 0.000,C 180.000} C_DIS
LIN {X 125.449,Y 115.685,Z 55.444,A 180.000,B 0.000,C 180.000} C_DIS
LIN {X 125.479,Y 115.758,Z 55.441,A 180.000,B 0.000,C 180.000} C_DIS
LIN {X 125.612,Y 116.129,Z 55.427,A 180.000,B 0.000,C 180.000} C_DIS
LIN {X 125.638,Y 116.203,Z 55.424,A 180.000,B 0.000,C 180.000} C_DIS
LIN {X 125.704,Y 116.430,Z 55.416,A 180.000,B 0.000,C 180.000} C_DIS
LIN {X 125.748,Y 116.581,Z 55.411,A 180.000,B 0.000,C 180.000} C_DIS
LIN {X 125.768,Y 116.657,Z 55.408,A 180.000,B 0.000,C 180.000} C_DIS
LIN {X 125.854,Y 117.042,Z 55.394,A 180.000,B 0.000,C 180.000} C_DIS
LIN {X 125.870,Y 117.119,Z 55.391,A 180.000,B 0.000,C 180.000} C_DIS
LIN {X 125.894,Y 117.274,Z 55.386,A 180.000,B 0.000,C 180.000} C_DIS
LIN {X 125.931,Y 117.508,Z 55.378,A 180.000,B 0.000,C 180.000} C_DIS
LIN {X 125.942,Y 117.586,Z 55.375,A 180.000,B 0.000,C 180.000} C_DIS
LIN {X 125.979,Y 117.978,Z 55.361,A 180.000,B 0.000,C 180.000} C_DIS
LIN {X 125.985,Y 118.056,Z 55.358,A 180.000,B 0.000,C 180.000} C_DIS
LIN {X 125.990,Y 118.214,Z 55.353,A 180.000,B 0.000,C 180.000} C_DIS
LIN {X 125.997,Y 118.450,Z 55.345,A 180.000,B 0.000,C 180.000} C_DIS
LIN {X 125.998,Y 118.529,Z 55.342,A 180.000,B 0.000,C 180.000} C_DIS
LIN {X 125.985,Y 118.922,Z 55.328,A 180.000,B 0.000,C 180.000} C_DIS
LIN {X 125.981,Y 119.001,Z 55.325,A 180.000,B 0.000,C 180.000} C_DIS
LIN {X 125.974,Y 119.079,Z 55.323,A 180.000,B 0.000,C 180.000} C_DIS
LIN {X 125.959,Y 119.236,Z 55.317,A 180.000,B 0.000,C 180.000} C_DIS
LIN {X 125.944,Y 119.393,Z 55.312,A 180.000,B 0.000,C 180.000} C_DIS
LIN {X 125.935,Y 119.471,Z 55.309,A 180.000,B 0.000,C 180.000} C_DIS
LIN {X 125.910,Y 119.627,Z 55.303,A 180.000,B 0.000,C 180.000} C_DIS
LIN {X 125.898,Y 119.705,Z 55.301,A 180.000,B 0.000,C 180.000} C_DIS
LIN {X 125.873,Y 119.860,Z 55.295,A 180.000,B 0.000,C 180.000} C_DIS
LIN {X 125.859,Y 119.938,Z 55.292,A 180.000,B 0.000,C 180.000} C_DIS
LIN {X 125.842,Y 120.014,Z 55.290,A 180.000,B 0.000,C 180.000} C_DIS
LIN {X 125.807,Y 120.168,Z 55.284,A 180.000,B 0.000,C 180.000} C_DIS
LIN {X 125.773,Y 120.322,Z 55.279,A 180.000,B 0.000,C 180.000} C_DIS
LIN {X 125.754,Y 120.398,Z 55.276,A 180.000,B 0.000,C 180.000} C_DIS
LIN {X 125.710,Y 120.549,Z 55.270,A 180.000,B 0.000,C 180.000} C_DIS
LIN {X 125.688,Y 120.625,Z 55.268,A 180.000,B 0.000,C 180.000} C_DIS
LIN {X 125.644,Y 120.776,Z 55.262,A 180.000,B 0.000,C 180.000} C_DIS
LIN {X 125.620,Y 120.851,Z 55.259,A 180.000,B 0.000,C 180.000} C_DIS
LIN {X 125.593,Y 120.925,Z 55.257,A 180.000,B 0.000,C 180.000} C_DIS
LIN {X 125.539,Y 121.074,Z 55.251,A 180.000,B 0.000,C 180.000} C_DIS
LIN {X 125.486,Y 121.222,Z 55.246,A 180.000,B 0.000,C 180.000} C_DIS
LIN {X 125.457,Y 121.295,Z 55.243,A 180.000,B 0.000,C 180.000} C_DIS
LIN {X 125.395,Y 121.440,Z 55.237,A 180.000,B 0.000,C 180.000} C_DIS
LIN {X 125.363,Y 121.512,Z 55.235,A 180.000,B 0.000,C 180.000} C_DIS
LIN {X 125.301,Y 121.656,Z 55.229,A 180.000,B 0.000,C 180.000} C_DIS
LIN {X 125.267,Y 121.728,Z 55.226,A 180.000,B 0.000,C 180.000} C_DIS
LIN {X 125.232,Y 121.798,Z 55.224,A 180.000,B 0.000,C 180.000} C_DIS
LIN {X 125.160,Y 121.938,Z 55.218,A 180.000,B 0.000,C 180.000} C_DIS
LIN {X 125.089,Y 122.079,Z 55.213,A 180.000,B 0.000,C 180.000} C_DIS
LIN {X 125.051,Y 122.147,Z 55.210,A 180.000,B 0.000,C 180.000} C_DIS
LIN {X 124.970,Y 122.283,Z 55.204,A 180.000,B 0.000,C 180.000} C_DIS
LIN {X 124.930,Y 122.351,Z 55.202,A 180.000,B 0.000,C 180.000} C_DIS
LIN {X 124.850,Y 122.486,Z 55.196,A 180.000,B 0.000,C 180.000} C_DIS
LIN {X 124.808,Y 122.553,Z 55.193,A 180.000,B 0.000,C 180.000} C_DIS
LIN {X 124.631,Y 122.813,Z 55.182,A 180.000,B 0.000,C 180.000} C_DIS
LIN {X 124.586,Y 122.878,Z 55.180,A 180.000,B 0.000,C 180.000} C_DIS
LIN {X 124.540,Y 122.942,Z 55.177,A 180.000,B 0.000,C 180.000} C_DIS
LIN {X 124.443,Y 123.067,Z 55.172,A 180.000,B 0.000,C 180.000} C_DIS
LIN {X 124.347,Y 123.191,Z 55.166,A 180.000,B 0.000,C 180.000} C_DIS
LIN {X 124.299,Y 123.253,Z 55.164,A 180.000,B 0.000,C 180.000} C_DIS
LIN {X 124.248,Y 123.314,Z 55.161,A 180.000,B 0.000,C 180.000} C_DIS
LIN {X 124.196,Y 123.373,Z 55.159,A 180.000,B 0.000,C 180.000} C_DIS
LIN {X 124.144,Y 123.432,Z 55.156,A 180.000,B 0.000,C 180.000} C_DIS
LIN {X 124.092,Y 123.491,Z 55.154,A 180.000,B 0.000,C 180.000} C_DIS
LIN {X 124.040,Y 123.550,Z 55.151,A 180.000,B 0.000,C 180.000} C_DIS
LIN {X 123.988,Y 123.609,Z 55.149,A 180.000,B 0.000,C 180.000} C_DIS
LIN {X 123.878,Y 123.722,Z 55.144,A 180.000,B 0.000,C 180.000} C_DIS
LIN {X 123.766,Y 123.833,Z 55.139,A 180.000,B 0.000,C 180.000} C_DIS
LIN {X 123.655,Y 123.945,Z 55.134,A 180.000,B 0.000,C 180.000} C_DIS
LIN {X 123.538,Y 124.050,Z 55.129,A 180.000,B 0.000,C 180.000} C_DIS
LIN {X 123.420,Y 124.154,Z 55.124,A 180.000,B 0.000,C 180.000} C_DIS
LIN {X 123.302,Y 124.259,Z 55.120,A 180.000,B 0.000,C 180.000} C_DIS
LIN {X 123.179,Y 124.357,Z 55.115,A 180.000,B 0.000,C 180.000} C_DIS
LIN {X 123.054,Y 124.453,Z 55.111,A 180.000,B 0.000,C 180.000} C_DIS
LIN {X 122.930,Y 124.550,Z 55.106,A 180.000,B 0.000,C 180.000} C_DIS
LIN {X 122.800,Y 124.640,Z 55.102,A 180.000,B 0.000,C 180.000} C_DIS
LIN {X 122.670,Y 124.728,Z 55.097,A 180.000,B 0.000,C 180.000} C_DIS
LIN {X 122.540,Y 124.817,Z 55.093,A 180.000,B 0.000,C 180.000} C_DIS
LIN {X 122.405,Y 124.898,Z 55.089,A 180.000,B 0.000,C 180.000} C_DIS
LIN {X 122.269,Y 124.978,Z 55.085,A 180.000,B 0.000,C 180.000} C_DIS
LIN {X 122.134,Y 125.059,Z 55.081,A 180.000,B 0.000,C 180.000} C_DIS
LIN {X 121.994,Y 125.131,Z 55.077,A 180.000,B 0.000,C 180.000} C_DIS
LIN {X 121.854,Y 125.203,Z 55.073,A 180.000,B 0.000,C 180.000} C_DIS
LIN {X 121.714,Y 125.274,Z 55.070,A 180.000,B 0.000,C 180.000} C_DIS
LIN {X 121.570,Y 125.338,Z 55.066,A 180.000,B 0.000,C 180.000} C_DIS
LIN {X 121.425,Y 125.401,Z 55.062,A 180.000,B 0.000,C 180.000} C_DIS
LIN {X 121.281,Y 125.464,Z 55.059,A 180.000,B 0.000,C 180.000} C_DIS
LIN {X 121.133,Y 125.518,Z 55.056,A 180.000,B 0.000,C 180.000} C_DIS
LIN {X 120.985,Y 125.572,Z 55.052,A 180.000,B 0.000,C 180.000} C_DIS
LIN {X 120.836,Y 125.625,Z 55.049,A 180.000,B 0.000,C 180.000} C_DIS
LIN {X 120.686,Y 125.670,Z 55.046,A 180.000,B 0.000,C 180.000} C_DIS
LIN {X 120.534,Y 125.714,Z 55.043,A 180.000,B 0.000,C 180.000} C_DIS
LIN {X 120.383,Y 125.758,Z 55.040,A 180.000,B 0.000,C 180.000} C_DIS
LIN {X 120.230,Y 125.793,Z 55.037,A 180.000,B 0.000,C 180.000} C_DIS
LIN {X 120.076,Y 125.828,Z 55.034,A 180.000,B 0.000,C 180.000} C_DIS
LIN {X 119.922,Y 125.862,Z 55.032,A 180.000,B 0.000,C 180.000} C_DIS
LIN {X 119.767,Y 125.888,Z 55.029,A 180.000,B 0.000,C 180.000} C_DIS
LIN {X 119.611,Y 125.913,Z 55.027,A 180.000,B 0.000,C 180.000} C_DIS
LIN {X 119.299,Y 125.953,Z 55.022,A 180.000,B 0.000,C 180.000} C_DIS
LIN {X 118.985,Y 125.983,Z 55.018,A 180.000,B 0.000,C 180.000} C_DIS
LIN {X 118.670,Y 125.993,Z 55.014,A 180.000,B 0.000,C 180.000} C_DIS
LIN {X 118.356,Y 125.994,Z 55.011,A 180.000,B 0.000,C 180.000} C_DIS
LIN {X 118.041,Y 125.984,Z 55.008,A 180.000,B 0.000,C 180.000} C_DIS
LIN {X 117.727,Y 125.955,Z 55.005,A 180.000,B 0.000,C 180.000} C_DIS
LIN {X 117.414,Y 125.917,Z 55.003,A 180.000,B 0.000,C 180.000} C_DIS
LIN {X 117.103,Y 125.867,Z 55.002,A 180.000,B 0.000,C 180.000} C_DIS
LIN {X 116.796,Y 125.799,Z 55.001,A 180.000,B 0.000,C 180.000} C_DIS
LIN {X 116.491,Y 125.721,Z 55.000,A 180.000,B 0.000,C 180.000} C_DIS
LIN {X 116.267,Y 125.656,Z 55.000,A 180.000,B 0.000,C 180.000} C_DIS
; Cutting Move Starts
LIN {X 116.204,Y 125.638,Z 55.000,A 180.000,B 0.000,C 180.000} C_DIS
LIN {X 116.025,Y 125.575,Z 55.000,A 180.000,B 0.000,C 180.000} C_DIS
LIN {X 115.816,Y 125.500,Z 55.000,A 180.000,B 0.000,C 180.000} C_DIS
LIN {X 115.667,Y 125.441,Z 55.000,A 180.000,B 0.000,C 180.000} C_DIS
LIN {X 115.310,Y 125.286,Z 55.000,A 180.000,B 0.000,C 180.000} C_DIS
LIN {X 115.131,Y 125.195,Z 55.000,A 180.000,B 0.000,C 180.000} C_DIS
LIN {X 114.952,Y 125.104,Z 55.000,A 180.000,B 0.000,C 180.000} C_DIS
LIN {X 114.774,Y 125.004,Z 55.000,A 180.000,B 0.000,C 180.000} C_DIS
LIN {X 114.595,Y 124.898,Z 55.000,A 180.000,B 0.000,C 180.000} C_DIS
LIN {X 114.416,Y 124.787,Z 55.000,A 180.000,B 0.000,C 180.000} C_DIS
LIN {X 114.150,Y 124.606,Z 55.000,A 180.000,B 0.000,C 180.000} C_DIS
LIN {X 114.058,Y 124.540,Z 55.000,A 180.000,B 0.000,C 180.000} C_DIS
LIN {X 113.880,Y 124.402,Z 55.000,A 180.000,B 0.000,C 180.000} C_DIS
LIN {X 113.701,Y 124.261,Z 55.000,A 180.000,B 0.000,C 180.000} C_DIS
LIN {X 113.484,Y 124.070,Z 55.000,A 180.000,B 0.000,C 180.000} C_DIS
LIN {X 113.343,Y 123.943,Z 55.000,A 180.000,B 0.000,C 180.000} C_DIS
LIN {X 113.112,Y 123.712,Z 55.000,A 180.000,B 0.000,C 180.000} C_DIS
LIN {X 112.986,Y 123.579,Z 55.000,A 180.000,B 0.000,C 180.000} C_DIS
LIN {X 112.788,Y 123.354,Z 55.000,A 180.000,B 0.000,C 180.000} C_DIS
LIN {X 112.641,Y 123.176,Z 55.000,A 180.000,B 0.000,C 180.000} C_DIS
LIN {X 112.450,Y 122.928,Z 55.000,A 180.000,B 0.000,C 180.000} C_DIS
LIN {X 112.373,Y 122.818,Z 55.000,A 180.000,B 0.000,C 180.000} C_DIS
LIN {X 112.251,Y 122.639,Z 55.000,A 180.000,B 0.000,C 180.000} C_DIS
LIN {X 112.135,Y 122.461,Z 55.000,A 180.000,B 0.000,C 180.000} C_DIS
LIN {X 112.029,Y 122.282,Z 55.000,A 180.000,B 0.000,C 180.000} C_DIS
LIN {X 111.924,Y 122.103,Z 55.000,A 180.000,B 0.000,C 180.000} C_DIS
LIN {X 111.734,Y 121.731,Z 55.000,A 180.000,B 0.000,C 180.000} C_DIS
LIN {X 111.660,Y 121.567,Z 55.000,A 180.000,B 0.000,C 180.000} C_DIS
LIN {X 111.556,Y 121.325,Z 55.000,A 180.000,B 0.000,C 180.000} C_DIS
LIN {X 111.509,Y 121.209,Z 55.000,A 180.000,B 0.000,C 180.000} C_DIS
LIN {X 111.377,Y 120.841,Z 55.000,A 180.000,B 0.000,C 180.000} C_DIS
LIN {X 111.326,Y 120.673,Z 55.000,A 180.000,B 0.000,C 180.000} C_DIS
LIN {X 111.274,Y 120.494,Z 55.000,A 180.000,B 0.000,C 180.000} C_DIS
LIN {X 111.226,Y 120.315,Z 55.000,A 180.000,B 0.000,C 180.000} C_DIS
LIN {X 111.146,Y 119.958,Z 55.000,A 180.000,B 0.000,C 180.000} C_DIS
LIN {X 111.114,Y 119.779,Z 55.000,A 180.000,B 0.000,C 180.000} C_DIS
LIN {X 111.086,Y 119.600,Z 55.000,A 180.000,B 0.000,C 180.000} C_DIS
LIN {X 111.059,Y 119.422,Z 55.000,A 180.000,B 0.000,C 180.000} C_DIS
LIN {X 111.019,Y 119.006,Z 55.000,A 180.000,B 0.000,C 180.000} C_DIS
LIN {X 111.013,Y 118.885,Z 55.000,A 180.000,B 0.000,C 180.000} C_DIS
LIN {X 111.002,Y 118.528,Z 55.000,A 180.000,B 0.000,C 180.000} C_DIS
LIN {X 111.006,Y 118.349,Z 55.000,A 180.000,B 0.000,C 180.000} C_DIS
LIN {X 111.012,Y 118.170,Z 55.000,A 180.000,B 0.000,C 180.000} C_DIS
LIN {X 111.019,Y 117.994,Z 55.000,A 180.000,B 0.000,C 180.000} C_DIS
LIN {X 111.053,Y 117.634,Z 55.000,A 180.000,B 0.000,C 180.000} C_DIS
LIN {X 111.077,Y 117.455,Z 55.000,A 180.000,B 0.000,C 180.000} C_DIS
LIN {X 111.134,Y 117.098,Z 55.000,A 180.000,B 0.000,C 180.000} C_DIS
LIN {X 111.173,Y 116.919,Z 55.000,A 180.000,B 0.000,C 180.000} C_DIS
LIN {X 111.213,Y 116.740,Z 55.000,A 180.000,B 0.000,C 180.000} C_DIS
LIN {X 111.258,Y 116.561,Z 55.000,A 180.000,B 0.000,C 180.000} C_DIS
LIN {X 111.362,Y 116.204,Z 55.000,A 180.000,B 0.000,C 180.000} C_DIS
LIN {X 111.377,Y 116.159,Z 55.000,A 180.000,B 0.000,C 180.000} C_DIS
LIN {X 111.489,Y 115.846,Z 55.000,A 180.000,B 0.000,C 180.000} C_DIS
LIN {X 111.556,Y 115.675,Z 55.000,A 180.000,B 0.000,C 180.000} C_DIS
LIN {X 111.714,Y 115.310,Z 55.000,A 180.000,B 0.000,C 180.000} C_DIS
LIN {X 111.734,Y 115.269,Z 55.000,A 180.000,B 0.000,C 180.000} C_DIS
LIN {X 111.913,Y 114.918,Z 55.000,A 180.000,B 0.000,C 180.000} C_DIS
LIN {X 111.996,Y 114.774,Z 55.000,A 180.000,B 0.000,C 180.000} C_DIS
LIN {X 112.102,Y 114.595,Z 55.000,A 180.000,B 0.000,C 180.000} C_DIS
LIN {X 112.213,Y 114.416,Z 55.000,A 180.000,B 0.000,C 180.000} C_DIS
LIN {X 112.335,Y 114.237,Z 55.000,A 180.000,B 0.000,C 180.000} C_DIS
LIN {X 112.450,Y 114.072,Z 55.000,A 180.000,B 0.000,C 180.000} C_DIS
LIN {X 112.628,Y 113.841,Z 55.000,A 180.000,B 0.000,C 180.000} C_DIS
LIN {X 112.739,Y 113.701,Z 55.000,A 180.000,B 0.000,C 180.000} C_DIS
LIN {X 112.986,Y 113.421,Z 55.000,A 180.000,B 0.000,C 180.000} C_DIS
LIN {X 113.057,Y 113.343,Z 55.000,A 180.000,B 0.000,C 180.000} C_DIS
LIN {X 113.343,Y 113.057,Z 55.000,A 180.000,B 0.000,C 180.000} C_DIS
LIN {X 113.421,Y 112.986,Z 55.000,A 180.000,B 0.000,C 180.000} C_DIS
LIN {X 113.701,Y 112.739,Z 55.000,A 180.000,B 0.000,C 180.000} C_DIS
LIN {X 113.841,Y 112.628,Z 55.000,A 180.000,B 0.000,C 180.000} C_DIS
LIN {X 114.072,Y 112.450,Z 55.000,A 180.000,B 0.000,C 180.000} C_DIS
LIN {X 114.237,Y 112.335,Z 55.000,A 180.000,B 0.000,C 180.000} C_DIS
LIN {X 114.416,Y 112.213,Z 55.000,A 180.000,B 0.000,C 180.000} C_DIS
LIN {X 114.595,Y 112.102,Z 55.000,A 180.000,B 0.000,C 180.000} C_DIS
LIN {X 114.774,Y 111.996,Z 55.000,A 180.000,B 0.000,C 180.000} C_DIS
LIN {X 114.918,Y 111.913,Z 55.000,A 180.000,B 0.000,C 180.000} C_DIS
LIN {X 115.269,Y 111.734,Z 55.000,A 180.000,B 0.000,C 180.000} C_DIS
LIN {X 115.310,Y 111.714,Z 55.000,A 180.000,B 0.000,C 180.000} C_DIS
LIN {X 115.675,Y 111.556,Z 55.000,A 180.000,B 0.000,C 180.000} C_DIS
LIN {X 115.846,Y 111.489,Z 55.000,A 180.000,B 0.000,C 180.000} C_DIS
LIN {X 116.159,Y 111.377,Z 55.000,A 180.000,B 0.000,C 180.000} C_DIS
LIN {X 116.204,Y 111.362,Z 55.000,A 180.000,B 0.000,C 180.000} C_DIS
LIN {X 116.561,Y 111.258,Z 55.000,A 180.000,B 0.000,C 180.000} C_DIS
LIN {X 116.740,Y 111.213,Z 55.000,A 180.000,B 0.000,C 180.000} C_DIS
LIN {X 116.919,Y 111.173,Z 55.000,A 180.000,B 0.000,C 180.000} C_DIS
LIN {X 117.098,Y 111.134,Z 55.000,A 180.000,B 0.000,C 180.000} C_DIS
LIN {X 117.455,Y 111.077,Z 55.000,A 180.000,B 0.000,C 180.000} C_DIS
LIN {X 117.634,Y 111.053,Z 55.000,A 180.000,B 0.000,C 180.000} C_DIS
LIN {X 117.994,Y 111.019,Z 55.000,A 180.000,B 0.000,C 180.000} C_DIS
LIN {X 118.170,Y 111.012,Z 55.000,A 180.000,B 0.000,C 180.000} C_DIS
LIN {X 118.349,Y 111.006,Z 55.000,A 180.000,B 0.000,C 180.000} C_DIS
LIN {X 118.528,Y 111.002,Z 55.000,A 180.000,B 0.000,C 180.000} C_DIS
LIN {X 118.885,Y 111.013,Z 55.000,A 180.000,B 0.000,C 180.000} C_DIS
LIN {X 119.006,Y 111.019,Z 55.000,A 180.000,B 0.000,C 180.000} C_DIS
LIN {X 119.422,Y 111.059,Z 55.000,A 180.000,B 0.000,C 180.000} C_DIS
LIN {X 119.600,Y 111.086,Z 55.000,A 180.000,B 0.000,C 180.000} C_DIS
LIN {X 119.779,Y 111.114,Z 55.000,A 180.000,B 0.000,C 180.000} C_DIS
LIN {X 119.958,Y 111.146,Z 55.000,A 180.000,B 0.000,C 180.000} C_DIS
LIN {X 120.315,Y 111.226,Z 55.000,A 180.000,B 0.000,C 180.000} C_DIS
LIN {X 120.494,Y 111.274,Z 55.000,A 180.000,B 0.000,C 180.000} C_DIS
LIN {X 120.673,Y 111.326,Z 55.000,A 180.000,B 0.000,C 180.000} C_DIS
LIN {X 120.841,Y 111.377,Z 55.000,A 180.000,B 0.000,C 180.000} C_DIS
LIN {X 121.209,Y 111.509,Z 55.000,A 180.000,B 0.000,C 180.000} C_DIS
LIN {X 121.325,Y 111.556,Z 55.000,A 180.000,B 0.000,C 180.000} C_DIS
LIN {X 121.567,Y 111.660,Z 55.000,A 180.000,B 0.000,C 180.000} C_DIS
LIN {X 121.731,Y 111.734,Z 55.000,A 180.000,B 0.000,C 180.000} C_DIS
LIN {X 122.103,Y 111.924,Z 55.000,A 180.000,B 0.000,C 180.000} C_DIS
LIN {X 122.282,Y 112.029,Z 55.000,A 180.000,B 0.000,C 180.000} C_DIS
LIN {X 122.461,Y 112.135,Z 55.000,A 180.000,B 0.000,C 180.000} C_DIS
LIN {X 122.639,Y 112.251,Z 55.000,A 180.000,B 0.000,C 180.000} C_DIS
LIN {X 122.818,Y 112.373,Z 55.000,A 180.000,B 0.000,C 180.000} C_DIS
LIN {X 122.928,Y 112.450,Z 55.000,A 180.000,B 0.000,C 180.000} C_DIS
LIN {X 123.176,Y 112.641,Z 55.000,A 180.000,B 0.000,C 180.000} C_DIS
LIN {X 123.354,Y 112.788,Z 55.000,A 180.000,B 0.000,C 180.000} C_DIS
LIN {X 123.579,Y 112.986,Z 55.000,A 180.000,B 0.000,C 180.000} C_DIS
LIN {X 123.712,Y 113.112,Z 55.000,A 180.000,B 0.000,C 180.000} C_DIS
LIN {X 123.943,Y 113.343,Z 55.000,A 180.000,B 0.000,C 180.000} C_DIS
LIN {X 124.070,Y 113.484,Z 55.000,A 180.000,B 0.000,C 180.000} C_DIS
LIN {X 124.261,Y 113.701,Z 55.000,A 180.000,B 0.000,C 180.000} C_DIS
LIN {X 124.402,Y 113.880,Z 55.000,A 180.000,B 0.000,C 180.000} C_DIS
LIN {X 124.540,Y 114.058,Z 55.000,A 180.000,B 0.000,C 180.000} C_DIS
LIN {X 124.606,Y 114.150,Z 55.000,A 180.000,B 0.000,C 180.000} C_DIS
LIN {X 124.787,Y 114.416,Z 55.000,A 180.000,B 0.000,C 180.000} C_DIS
LIN {X 124.898,Y 114.595,Z 55.000,A 180.000,B 0.000,C 180.000} C_DIS
LIN {X 125.004,Y 114.774,Z 55.000,A 180.000,B 0.000,C 180.000} C_DIS
LIN {X 125.104,Y 114.952,Z 55.000,A 180.000,B 0.000,C 180.000} C_DIS
LIN {X 125.195,Y 115.131,Z 55.000,A 180.000,B 0.000,C 180.000} C_DIS
LIN {X 125.286,Y 115.310,Z 55.000,A 180.000,B 0.000,C 180.000} C_DIS
LIN {X 125.441,Y 115.667,Z 55.000,A 180.000,B 0.000,C 180.000} C_DIS
LIN {X 125.500,Y 115.816,Z 55.000,A 180.000,B 0.000,C 180.000} C_DIS
LIN {X 125.575,Y 116.025,Z 55.000,A 180.000,B 0.000,C 180.000} C_DIS
LIN {X 125.638,Y 116.204,Z 55.000,A 180.000,B 0.000,C 180.000} C_DIS
LIN {X 125.742,Y 116.561,Z 55.000,A 180.000,B 0.000,C 180.000} C_DIS
LIN {X 125.787,Y 116.740,Z 55.000,A 180.000,B 0.000,C 180.000} C_DIS
LIN {X 125.857,Y 117.056,Z 55.000,A 180.000,B 0.000,C 180.000} C_DIS
LIN {X 125.866,Y 117.098,Z 55.000,A 180.000,B 0.000,C 180.000} C_DIS
LIN {X 125.923,Y 117.455,Z 55.000,A 180.000,B 0.000,C 180.000} C_DIS
LIN {X 125.947,Y 117.634,Z 55.000,A 180.000,B 0.000,C 180.000} C_DIS
LIN {X 125.980,Y 117.991,Z 55.000,A 180.000,B 0.000,C 180.000} C_DIS
LIN {X 125.988,Y 118.170,Z 55.000,A 180.000,B 0.000,C 180.000} C_DIS
LIN {X 125.994,Y 118.349,Z 55.000,A 180.000,B 0.000,C 180.000} C_DIS
LIN {X 125.998,Y 118.528,Z 55.000,A 180.000,B 0.000,C 180.000} C_DIS
LIN {X 125.987,Y 118.885,Z 55.000,A 180.000,B 0.000,C 180.000} C_DIS
LIN {X 125.975,Y 119.064,Z 55.000,A 180.000,B 0.000,C 180.000} C_DIS
LIN {X 125.941,Y 119.422,Z 55.000,A 180.000,B 0.000,C 180.000} C_DIS
LIN {X 125.914,Y 119.600,Z 55.000,A 180.000,B 0.000,C 180.000} C_DIS
LIN {X 125.886,Y 119.779,Z 55.000,A 180.000,B 0.000,C 180.000} C_DIS
LIN {X 125.857,Y 119.944,Z 55.000,A 180.000,B 0.000,C 180.000} C_DIS
LIN {X 125.774,Y 120.315,Z 55.000,A 180.000,B 0.000,C 180.000} C_DIS
LIN {X 125.726,Y 120.494,Z 55.000,A 180.000,B 0.000,C 180.000} C_DIS
LIN {X 125.674,Y 120.673,Z 55.000,A 180.000,B 0.000,C 180.000} C_DIS
LIN {X 125.619,Y 120.852,Z 55.000,A 180.000,B 0.000,C 180.000} C_DIS
LIN {X 125.491,Y 121.209,Z 55.000,A 180.000,B 0.000,C 180.000} C_DIS
LIN {X 125.417,Y 121.388,Z 55.000,A 180.000,B 0.000,C 180.000} C_DIS
LIN {X 125.321,Y 121.610,Z 55.000,A 180.000,B 0.000,C 180.000} C_DIS
LIN {X 125.258,Y 121.746,Z 55.000,A 180.000,B 0.000,C 180.000} C_DIS
LIN {X 125.076,Y 122.103,Z 55.000,A 180.000,B 0.000,C 180.000} C_DIS
LIN {X 124.971,Y 122.282,Z 55.000,A 180.000,B 0.000,C 180.000} C_DIS
LIN {X 124.865,Y 122.461,Z 55.000,A 180.000,B 0.000,C 180.000} C_DIS
LIN {X 124.785,Y 122.587,Z 55.000,A 180.000,B 0.000,C 180.000} C_DIS
LIN {X 124.606,Y 122.850,Z 55.000,A 180.000,B 0.000,C 180.000} C_DIS
LIN {X 124.497,Y 122.997,Z 55.000,A 180.000,B 0.000,C 180.000} C_DIS
LIN {X 124.359,Y 123.176,Z 55.000,A 180.000,B 0.000,C 180.000} C_DIS
LIN {X 124.248,Y 123.313,Z 55.000,A 180.000,B 0.000,C 180.000} C_DIS
LIN {X 124.055,Y 123.533,Z 55.000,A 180.000,B 0.000,C 180.000} C_DIS
LIN {X 123.891,Y 123.709,Z 55.000,A 180.000,B 0.000,C 180.000} C_DIS
LIN {X 123.709,Y 123.891,Z 55.000,A 180.000,B 0.000,C 180.000} C_DIS
LIN {X 123.533,Y 124.055,Z 55.000,A 180.000,B 0.000,C 180.000} C_DIS
LIN {X 123.313,Y 124.248,Z 55.000,A 180.000,B 0.000,C 180.000} C_DIS
LIN {X 123.176,Y 124.359,Z 55.000,A 180.000,B 0.000,C 180.000} C_DIS
LIN {X 122.997,Y 124.497,Z 55.000,A 180.000,B 0.000,C 180.000} C_DIS
LIN {X 122.850,Y 124.606,Z 55.000,A 180.000,B 0.000,C 180.000} C_DIS
LIN {X 122.587,Y 124.785,Z 55.000,A 180.000,B 0.000,C 180.000} C_DIS
LIN {X 122.461,Y 124.865,Z 55.000,A 180.000,B 0.000,C 180.000} C_DIS
LIN {X 122.282,Y 124.971,Z 55.000,A 180.000,B 0.000,C 180.000} C_DIS
LIN {X 122.103,Y 125.076,Z 55.000,A 180.000,B 0.000,C 180.000} C_DIS
LIN {X 121.746,Y 125.258,Z 55.000,A 180.000,B 0.000,C 180.000} C_DIS
LIN {X 121.610,Y 125.321,Z 55.000,A 180.000,B 0.000,C 180.000} C_DIS
LIN {X 121.388,Y 125.417,Z 55.000,A 180.000,B 0.000,C 180.000} C_DIS
LIN {X 121.209,Y 125.491,Z 55.000,A 180.000,B 0.000,C 180.000} C_DIS
LIN {X 120.852,Y 125.619,Z 55.000,A 180.000,B 0.000,C 180.000} C_DIS
LIN {X 120.673,Y 125.674,Z 55.000,A 180.000,B 0.000,C 180.000} C_DIS
LIN {X 120.494,Y 125.726,Z 55.000,A 180.000,B 0.000,C 180.000} C_DIS
LIN {X 120.315,Y 125.774,Z 55.000,A 180.000,B 0.000,C 180.000} C_DIS
LIN {X 119.944,Y 125.857,Z 55.000,A 180.000,B 0.000,C 180.000} C_DIS
LIN {X 119.779,Y 125.886,Z 55.000,A 180.000,B 0.000,C 180.000} C_DIS
LIN {X 119.600,Y 125.914,Z 55.000,A 180.000,B 0.000,C 180.000} C_DIS
LIN {X 119.422,Y 125.941,Z 55.000,A 180.000,B 0.000,C 180.000} C_DIS
LIN {X 119.064,Y 125.975,Z 55.000,A 180.000,B 0.000,C 180.000} C_DIS
LIN {X 118.885,Y 125.987,Z 55.000,A 180.000,B 0.000,C 180.000} C_DIS
LIN {X 118.528,Y 125.998,Z 55.000,A 180.000,B 0.000,C 180.000} C_DIS
LIN {X 118.349,Y 125.994,Z 55.000,A 180.000,B 0.000,C 180.000} C_DIS
LIN {X 118.170,Y 125.988,Z 55.000,A 180.000,B 0.000,C 180.000} C_DIS
LIN {X 117.991,Y 125.980,Z 55.000,A 180.000,B 0.000,C 180.000} C_DIS
LIN {X 117.634,Y 125.947,Z 55.000,A 180.000,B 0.000,C 180.000} C_DIS
LIN {X 117.455,Y 125.923,Z 55.000,A 180.000,B 0.000,C 180.000} C_DIS
LIN {X 117.098,Y 125.866,Z 55.000,A 180.000,B 0.000,C 180.000} C_DIS
LIN {X 117.056,Y 125.857,Z 55.000,A 180.000,B 0.000,C 180.000} C_DIS
LIN {X 116.740,Y 125.787,Z 55.000,A 180.000,B 0.000,C 180.000} C_DIS
LIN {X 116.561,Y 125.742,Z 55.000,A 180.000,B 0.000,C 180.000} C_DIS
LIN {X 116.267,Y 125.656,Z 55.000,A 180.000,B 0.000,C 180.000} C_DIS
; Link Move Starts
LIN {X 115.969,Y 125.555,Z 55.000,A 180.000,B 0.000,C 180.000} C_DIS
LIN {X 115.674,Y 125.444,Z 54.999,A 180.000,B 0.000,C 180.000} C_DIS
LIN {X 115.385,Y 125.319,Z 54.998,A 180.000,B 0.000,C 180.000} C_DIS
LIN {X 115.102,Y 125.181,Z 54.996,A 180.000,B 0.000,C 180.000} C_DIS
LIN {X 114.823,Y 125.033,Z 54.994,A 180.000,B 0.000,C 180.000} C_DIS
LIN {X 114.552,Y 124.873,Z 54.991,A 180.000,B 0.000,C 180.000} C_DIS
LIN {X 114.289,Y 124.700,Z 54.988,A 180.000,B 0.000,C 180.000} C_DIS
LIN {X 114.031,Y 124.519,Z 54.985,A 180.000,B 0.000,C 180.000} C_DIS
LIN {X 113.782,Y 124.326,Z 54.981,A 180.000,B 0.000,C 180.000} C_DIS
LIN {X 113.543,Y 124.122,Z 54.977,A 180.000,B 0.000,C 180.000} C_DIS
LIN {X 113.310,Y 123.910,Z 54.972,A 180.000,B 0.000,C 180.000} C_DIS
LIN {X 113.199,Y 123.798,Z 54.969,A 180.000,B 0.000,C 180.000} C_DIS
LIN {X 113.087,Y 123.687,Z 54.967,A 180.000,B 0.000,C 180.000} C_DIS
LIN {X 112.980,Y 123.572,Z 54.964,A 180.000,B 0.000,C 180.000} C_DIS
LIN {X 112.875,Y 123.454,Z 54.961,A 180.000,B 0.000,C 180.000} C_DIS
LIN {X 112.771,Y 123.336,Z 54.959,A 180.000,B 0.000,C 180.000} C_DIS
LIN {X 112.671,Y 123.214,Z 54.956,A 180.000,B 0.000,C 180.000} C_DIS
LIN {X 112.575,Y 123.090,Z 54.952,A 180.000,B 0.000,C 180.000} C_DIS
LIN {X 112.478,Y 122.965,Z 54.949,A 180.000,B 0.000,C 180.000} C_DIS
LIN {X 112.386,Y 122.838,Z 54.946,A 180.000,B 0.000,C 180.000} C_DIS
LIN {X 112.297,Y 122.707,Z 54.943,A 180.000,B 0.000,C 180.000} C_DIS
LIN {X 112.209,Y 122.577,Z 54.939,A 180.000,B 0.000,C 180.000} C_DIS
LIN {X 112.125,Y 122.444,Z 54.936,A 180.000,B 0.000,C 180.000} C_DIS
LIN {X 112.045,Y 122.308,Z 54.932,A 180.000,B 0.000,C 180.000} C_DIS
LIN {X 111.964,Y 122.173,Z 54.928,A 180.000,B 0.000,C 180.000} C_DIS
LIN {X 111.889,Y 122.034,Z 54.925,A 180.000,B 0.000,C 180.000} C_DIS
LIN {X 111.817,Y 121.894,Z 54.921,A 180.000,B 0.000,C 180.000} C_DIS
LIN {X 111.746,Y 121.754,Z 54.917,A 180.000,B 0.000,C 180.000} C_DIS
LIN {X 111.680,Y 121.611,Z 54.913,A 180.000,B 0.000,C 180.000} C_DIS
LIN {X 111.617,Y 121.466,Z 54.909,A 180.000,B 0.000,C 180.000} C_DIS
LIN {X 111.554,Y 121.322,Z 54.905,A 180.000,B 0.000,C 180.000} C_DIS
LIN {X 111.497,Y 121.175,Z 54.900,A 180.000,B 0.000,C 180.000} C_DIS
LIN {X 111.444,Y 121.027,Z 54.896,A 180.000,B 0.000,C 180.000} C_DIS
LIN {X 111.390,Y 120.879,Z 54.892,A 180.000,B 0.000,C 180.000} C_DIS
LIN {X 111.343,Y 120.729,Z 54.887,A 180.000,B 0.000,C 180.000} C_DIS
LIN {X 111.299,Y 120.578,Z 54.883,A 180.000,B 0.000,C 180.000} C_DIS
LIN {X 111.255,Y 120.426,Z 54.878,A 180.000,B 0.000,C 180.000} C_DIS
LIN {X 111.216,Y 120.274,Z 54.873,A 180.000,B 0.000,C 180.000} C_DIS
LIN {X 111.182,Y 120.120,Z 54.869,A 180.000,B 0.000,C 180.000} C_DIS
LIN {X 111.148,Y 119.966,Z 54.864,A 180.000,B 0.000,C 180.000} C_DIS
LIN {X 111.119,Y 119.811,Z 54.859,A 180.000,B 0.000,C 180.000} C_DIS
LIN {X 111.095,Y 119.656,Z 54.854,A 180.000,B 0.000,C 180.000} C_DIS
LIN {X 111.082,Y 119.578,Z 54.851,A 180.000,B 0.000,C 180.000} C_DIS
LIN {X 111.070,Y 119.500,Z 54.849,A 180.000,B 0.000,C 180.000} C_DIS
LIN {X 111.059,Y 119.422,Z 54.846,A 180.000,B 0.000,C 180.000} C_DIS
LIN {X 111.051,Y 119.344,Z 54.844,A 180.000,B 0.000,C 180.000} C_DIS
LIN {X 111.044,Y 119.265,Z 54.841,A 180.000,B 0.000,C 180.000} C_DIS
LIN {X 111.036,Y 119.187,Z 54.839,A 180.000,B 0.000,C 180.000} C_DIS
LIN {X 111.029,Y 119.109,Z 54.836,A 180.000,B 0.000,C 180.000} C_DIS
LIN {X 111.022,Y 119.030,Z 54.833,A 180.000,B 0.000,C 180.000} C_DIS
LIN {X 111.015,Y 118.952,Z 54.831,A 180.000,B 0.000,C 180.000} C_DIS
LIN {X 111.013,Y 118.873,Z 54.828,A 180.000,B 0.000,C 180.000} C_DIS
LIN {X 111.008,Y 118.716,Z 54.823,A 180.000,B 0.000,C 180.000} C_DIS
LIN {X 111.003,Y 118.558,Z 54.817,A 180.000,B 0.000,C 180.000} C_DIS
LIN {X 111.002,Y 118.479,Z 54.815,A 180.000,B 0.000,C 180.000} C_DIS
LIN {X 111.007,Y 118.322,Z 54.809,A 180.000,B 0.000,C 180.000} C_DIS
LIN {X 111.009,Y 118.243,Z 54.806,A 180.000,B 0.000,C 180.000} C_DIS
LIN {X 111.014,Y 118.086,Z 54.801,A 180.000,B 0.000,C 180.000} C_DIS
LIN {X 111.018,Y 118.007,Z 54.798,A 180.000,B 0.000,C 180.000} C_DIS
LIN {X 111.026,Y 117.929,Z 54.796,A 180.000,B 0.000,C 180.000} C_DIS
LIN {X 111.040,Y 117.772,Z 54.790,A 180.000,B 0.000,C 180.000} C_DIS
LIN {X 111.055,Y 117.615,Z 54.785,A 180.000,B 0.000,C 180.000} C_DIS
LIN {X 111.064,Y 117.537,Z 54.782,A 180.000,B 0.000,C 180.000} C_DIS
LIN {X 111.089,Y 117.381,Z 54.776,A 180.000,B 0.000,C 180.000} C_DIS
LIN {X 111.101,Y 117.303,Z 54.774,A 180.000,B 0.000,C 180.000} C_DIS
LIN {X 111.126,Y 117.148,Z 54.768,A 180.000,B 0.000,C 180.000} C_DIS
LIN {X 111.140,Y 117.070,Z 54.765,A 180.000,B 0.000,C 180.000} C_DIS
LIN {X 111.157,Y 116.994,Z 54.763,A 180.000,B 0.000,C 180.000} C_DIS
LIN {X 111.191,Y 116.840,Z 54.757,A 180.000,B 0.000,C 180.000} C_DIS
LIN {X 111.225,Y 116.686,Z 54.752,A 180.000,B 0.000,C 180.000} C_DIS
LIN {X 111.244,Y 116.610,Z 54.749,A 180.000,B 0.000,C 180.000} C_DIS
LIN {X 111.288,Y 116.458,Z 54.743,A 180.000,B 0.000,C 180.000} C_DIS
LIN {X 111.310,Y 116.383,Z 54.741,A 180.000,B 0.000,C 180.000} C_DIS
LIN {X 111.354,Y 116.232,Z 54.735,A 180.000,B 0.000,C 180.000} C_DIS
LIN {X 111.378,Y 116.156,Z 54.732,A 180.000,B 0.000,C 180.000} C_DIS
LIN {X 111.404,Y 116.082,Z 54.730,A 180.000,B 0.000,C 180.000} C_DIS
LIN {X 111.458,Y 115.934,Z 54.724,A 180.000,B 0.000,C 180.000} C_DIS
LIN {X 111.511,Y 115.786,Z 54.719,A 180.000,B 0.000,C 180.000} C_DIS
LIN {X 111.540,Y 115.712,Z 54.716,A 180.000,B 0.000,C 180.000} C_DIS
LIN {X 111.602,Y 115.568,Z 54.710,A 180.000,B 0.000,C 180.000} C_DIS
LIN {X 111.633,Y 115.496,Z 54.708,A 180.000,B 0.000,C 180.000} C_DIS
LIN {X 111.696,Y 115.351,Z 54.702,A 180.000,B 0.000,C 180.000} C_DIS
LIN {X 111.729,Y 115.280,Z 54.699,A 180.000,B 0.000,C 180.000} C_DIS
LIN {X 111.765,Y 115.209,Z 54.697,A 180.000,B 0.000,C 180.000} C_DIS
LIN {X 111.836,Y 115.069,Z 54.691,A 180.000,B 0.000,C 180.000} C_DIS
LIN {X 111.908,Y 114.929,Z 54.686,A 180.000,B 0.000,C 180.000} C_DIS
LIN {X 111.945,Y 114.860,Z 54.683,A 180.000,B 0.000,C 180.000} C_DIS
LIN {X 112.025,Y 114.724,Z 54.677,A 180.000,B 0.000,C 180.000} C_DIS
LIN {X 112.066,Y 114.656,Z 54.675,A 180.000,B 0.000,C 180.000} C_DIS
LIN {X 112.146,Y 114.521,Z 54.669,A 180.000,B 0.000,C 180.000} C_DIS
LIN {X 112.188,Y 114.454,Z 54.666,A 180.000,B 0.000,C 180.000} C_DIS
LIN {X 112.276,Y 114.324,Z 54.661,A 180.000,B 0.000,C 180.000} C_DIS
LIN {X 112.409,Y 114.128,Z 54.653,A 180.000,B 0.000,C 180.000} C_DIS
LIN {X 112.455,Y 114.064,Z 54.650,A 180.000,B 0.000,C 180.000} C_DIS
LIN {X 112.696,Y 113.753,Z 54.636,A 180.000,B 0.000,C 180.000} C_DIS
LIN {X 112.746,Y 113.693,Z 54.633,A 180.000,B 0.000,C 180.000} C_DIS
LIN {X 112.851,Y 113.574,Z 54.628,A 180.000,B 0.000,C 180.000} C_DIS
LIN {X 113.007,Y 113.397,Z 54.620,A 180.000,B 0.000,C 180.000} C_DIS
LIN {X 113.061,Y 113.340,Z 54.617,A 180.000,B 0.000,C 180.000} C_DIS
LIN {X 113.339,Y 113.061,Z 54.603,A 180.000,B 0.000,C 180.000} C_DIS
LIN {X 113.397,Y 113.007,Z 54.600,A 180.000,B 0.000,C 180.000} C_DIS
LIN {X 113.692,Y 112.747,Z 54.587,A 180.000,B 0.000,C 180.000} C_DIS
LIN {X 113.753,Y 112.697,Z 54.584,A 180.000,B 0.000,C 180.000} C_DIS
LIN {X 114.064,Y 112.456,Z 54.570,A 180.000,B 0.000,C 180.000} C_DIS
LIN {X 114.128,Y 112.409,Z 54.567,A 180.000,B 0.000,C 180.000} C_DIS
LIN {X 114.453,Y 112.188,Z 54.554,A 180.000,B 0.000,C 180.000} C_DIS
LIN {X 114.520,Y 112.146,Z 54.551,A 180.000,B 0.000,C 180.000} C_DIS
LIN {X 114.859,Y 111.946,Z 54.537,A 180.000,B 0.000,C 180.000} C_DIS
LIN {X 114.928,Y 111.908,Z 54.534,A 180.000,B 0.000,C 180.000} C_DIS
LIN {X 115.279,Y 111.729,Z 54.521,A 180.000,B 0.000,C 180.000} C_DIS
LIN {X 115.350,Y 111.696,Z 54.518,A 180.000,B 0.000,C 180.000} C_DIS
LIN {X 115.712,Y 111.540,Z 54.504,A 180.000,B 0.000,C 180.000} C_DIS
LIN {X 115.785,Y 111.511,Z 54.501,A 180.000,B 0.000,C 180.000} C_DIS
LIN {X 116.156,Y 111.378,Z 54.488,A 180.000,B 0.000,C 180.000} C_DIS
LIN {X 116.231,Y 111.354,Z 54.485,A 180.000,B 0.000,C 180.000} C_DIS
LIN {X 116.609,Y 111.244,Z 54.471,A 180.000,B 0.000,C 180.000} C_DIS
LIN {X 116.685,Y 111.226,Z 54.468,A 180.000,B 0.000,C 180.000} C_DIS
LIN {X 117.070,Y 111.140,Z 54.455,A 180.000,B 0.000,C 180.000} C_DIS
LIN {X 117.147,Y 111.126,Z 54.452,A 180.000,B 0.000,C 180.000} C_DIS
LIN {X 117.536,Y 111.064,Z 54.438,A 180.000,B 0.000,C 180.000} C_DIS
LIN {X 117.614,Y 111.055,Z 54.435,A 180.000,B 0.000,C 180.000} C_DIS
LIN {X 118.006,Y 111.018,Z 54.422,A 180.000,B 0.000,C 180.000} C_DIS
LIN {X 118.085,Y 111.014,Z 54.419,A 180.000,B 0.000,C 180.000} C_DIS
LIN {X 118.479,Y 111.002,Z 54.405,A 180.000,B 0.000,C 180.000} C_DIS
LIN {X 118.557,Y 111.003,Z 54.402,A 180.000,B 0.000,C 180.000} C_DIS
LIN {X 118.715,Y 111.008,Z 54.397,A 180.000,B 0.000,C 180.000} C_DIS
LIN {X 118.951,Y 111.015,Z 54.389,A 180.000,B 0.000,C 180.000} C_DIS
LIN {X 119.029,Y 111.022,Z 54.386,A 180.000,B 0.000,C 180.000} C_DIS
LIN {X 119.421,Y 111.059,Z 54.372,A 180.000,B 0.000,C 180.000} C_DIS
LIN {X 119.499,Y 111.070,Z 54.369,A 180.000,B 0.000,C 180.000} C_DIS
LIN {X 119.655,Y 111.094,Z 54.364,A 180.000,B 0.000,C 180.000} C_DIS
LIN {X 119.888,Y 111.131,Z 54.356,A 180.000,B 0.000,C 180.000} C_DIS
LIN {X 119.965,Y 111.148,Z 54.353,A 180.000,B 0.000,C 180.000} C_DIS
LIN {X 120.350,Y 111.233,Z 54.339,A 180.000,B 0.000,C 180.000} C_DIS
LIN {X 120.426,Y 111.254,Z 54.336,A 180.000,B 0.000,C 180.000} C_DIS
LIN {X 120.501,Y 111.276,Z 54.334,A 180.000,B 0.000,C 180.000} C_DIS
LIN {X 120.652,Y 111.320,Z 54.328,A 180.000,B 0.000,C 180.000} C_DIS
LIN {X 120.804,Y 111.364,Z 54.323,A 180.000,B 0.000,C 180.000} C_DIS
LIN {X 120.878,Y 111.390,Z 54.320,A 180.000,B 0.000,C 180.000} C_DIS
LIN {X 121.026,Y 111.444,Z 54.314,A 180.000,B 0.000,C 180.000} C_DIS
LIN {X 121.100,Y 111.470,Z 54.312,A 180.000,B 0.000,C 180.000} C_DIS
LIN {X 121.249,Y 111.524,Z 54.306,A 180.000,B 0.000,C 180.000} C_DIS
LIN {X 121.321,Y 111.554,Z 54.303,A 180.000,B 0.000,C 180.000} C_DIS
LIN {X 121.393,Y 111.585,Z 54.301,A 180.000,B 0.000,C 180.000} C_DIS
LIN {X 121.538,Y 111.648,Z 54.295,A 180.000,B 0.000,C 180.000} C_DIS
LIN {X 121.683,Y 111.710,Z 54.290,A 180.000,B 0.000,C 180.000} C_DIS
LIN {X 121.753,Y 111.746,Z 54.287,A 180.000,B 0.000,C 180.000} C_DIS
LIN {X 121.893,Y 111.817,Z 54.281,A 180.000,B 0.000,C 180.000} C_DIS
LIN {X 121.964,Y 111.853,Z 54.279,A 180.000,B 0.000,C 180.000} C_DIS
LIN {X 122.104,Y 111.924,Z 54.273,A 180.000,B 0.000,C 180.000} C_DIS
LIN {X 122.172,Y 111.964,Z 54.270,A 180.000,B 0.000,C 180.000} C_DIS
LIN {X 122.240,Y 112.004,Z 54.268,A 180.000,B 0.000,C 180.000} C_DIS
LIN {X 122.375,Y 112.084,Z 54.262,A 180.000,B 0.000,C 180.000} C_DIS
LIN {X 122.511,Y 112.164,Z 54.257,A 180.000,B 0.000,C 180.000} C_DIS
LIN {X 122.576,Y 112.208,Z 54.254,A 180.000,B 0.000,C 180.000} C_DIS
LIN {X 122.707,Y 112.297,Z 54.248,A 180.000,B 0.000,C 180.000} C_DIS
LIN {X 122.772,Y 112.341,Z 54.246,A 180.000,B 0.000,C 180.000} C_DIS
LIN {X 122.902,Y 112.430,Z 54.240,A 180.000,B 0.000,C 180.000} C_DIS
LIN {X 122.965,Y 112.478,Z 54.237,A 180.000,B 0.000,C 180.000} C_DIS
LIN {X 123.027,Y 112.526,Z 54.235,A 180.000,B 0.000,C 180.000} C_DIS
LIN {X 123.151,Y 112.622,Z 54.229,A 180.000,B 0.000,C 180.000} C_DIS
LIN {X 123.276,Y 112.719,Z 54.224,A 180.000,B 0.000,C 180.000} C_DIS
LIN {X 123.335,Y 112.771,Z 54.221,A 180.000,B 0.000,C 180.000} C_DIS
LIN {X 123.453,Y 112.875,Z 54.215,A 180.000,B 0.000,C 180.000} C_DIS
LIN {X 123.512,Y 112.927,Z 54.213,A 180.000,B 0.000,C 180.000} C_DIS
LIN {X 123.630,Y 113.031,Z 54.207,A 180.000,B 0.000,C 180.000} C_DIS
LIN {X 123.686,Y 113.087,Z 54.204,A 180.000,B 0.000,C 180.000} C_DIS
LIN {X 123.742,Y 113.142,Z 54.202,A 180.000,B 0.000,C 180.000} C_DIS
LIN {X 123.853,Y 113.254,Z 54.196,A 180.000,B 0.000,C 180.000} C_DIS
LIN {X 123.965,Y 113.365,Z 54.191,A 180.000,B 0.000,C 180.000} C_DIS
LIN {X 124.017,Y 113.424,Z 54.188,A 180.000,B 0.000,C 180.000} C_DIS
LIN {X 124.121,Y 113.542,Z 54.182,A 180.000,B 0.000,C 180.000} C_DIS
LIN {X 124.225,Y 113.660,Z 54.177,A 180.000,B 0.000,C 180.000} C_DIS
LIN {X 124.277,Y 113.720,Z 54.174,A 180.000,B 0.000,C 180.000} C_DIS
LIN {X 124.326,Y 113.782,Z 54.172,A 180.000,B 0.000,C 180.000} C_DIS
LIN {X 124.422,Y 113.906,Z 54.166,A 180.000,B 0.000,C 180.000} C_DIS
LIN {X 124.470,Y 113.968,Z 54.164,A 180.000,B 0.000,C 180.000} C_DIS
LIN {X 124.519,Y 114.031,Z 54.161,A 180.000,B 0.000,C 180.000} C_DIS
LIN {X 124.567,Y 114.093,Z 54.159,A 180.000,B 0.000,C 180.000} C_DIS
LIN {X 124.611,Y 114.158,Z 54.156,A 180.000,B 0.000,C 180.000} C_DIS
LIN {X 124.656,Y 114.223,Z 54.154,A 180.000,B 0.000,C 180.000} C_DIS
LIN {X 124.700,Y 114.288,Z 54.151,A 180.000,B 0.000,C 180.000} C_DIS
LIN {X 124.744,Y 114.353,Z 54.149,A 180.000,B 0.000,C 180.000} C_DIS
LIN {X 124.833,Y 114.484,Z 54.144,A 180.000,B 0.000,C 180.000} C_DIS
LIN {X 124.913,Y 114.619,Z 54.139,A 180.000,B 0.000,C 180.000} C_DIS
LIN {X 124.993,Y 114.755,Z 54.134,A 180.000,B 0.000,C 180.000} C_DIS
LIN {X 125.073,Y 114.891,Z 54.129,A 180.000,B 0.000,C 180.000} C_DIS
LIN {X 125.144,Y 115.031,Z 54.124,A 180.000,B 0.000,C 180.000} C_DIS
LIN {X 125.216,Y 115.171,Z 54.120,A 180.000,B 0.000,C 180.000} C_DIS
LIN {X 125.287,Y 115.312,Z 54.115,A 180.000,B 0.000,C 180.000} C_DIS
LIN {X 125.350,Y 115.456,Z 54.111,A 180.000,B 0.000,C 180.000} C_DIS
LIN {X 125.412,Y 115.601,Z 54.106,A 180.000,B 0.000,C 180.000} C_DIS
LIN {X 125.474,Y 115.746,Z 54.102,A 180.000,B 0.000,C 180.000} C_DIS
LIN {X 125.528,Y 115.894,Z 54.097,A 180.000,B 0.000,C 180.000} C_DIS
LIN {X 125.581,Y 116.042,Z 54.093,A 180.000,B 0.000,C 180.000} C_DIS
LIN {X 125.634,Y 116.190,Z 54.089,A 180.000,B 0.000,C 180.000} C_DIS
LIN {X 125.678,Y 116.342,Z 54.085,A 180.000,B 0.000,C 180.000} C_DIS
LIN {X 125.722,Y 116.493,Z 54.081,A 180.000,B 0.000,C 180.000} C_DIS
LIN {X 125.765,Y 116.644,Z 54.077,A 180.000,B 0.000,C 180.000} C_DIS
LIN {X 125.800,Y 116.798,Z 54.073,A 180.000,B 0.000,C 180.000} C_DIS
LIN {X 125.834,Y 116.952,Z 54.070,A 180.000,B 0.000,C 180.000} C_DIS
LIN {X 125.868,Y 117.106,Z 54.066,A 180.000,B 0.000,C 180.000} C_DIS
LIN {X 125.892,Y 117.261,Z 54.062,A 180.000,B 0.000,C 180.000} C_DIS
LIN {X 125.917,Y 117.417,Z 54.059,A 180.000,B 0.000,C 180.000} C_DIS
LIN {X 125.941,Y 117.573,Z 54.056,A 180.000,B 0.000,C 180.000} C_DIS
LIN {X 125.956,Y 117.729,Z 54.052,A 180.000,B 0.000,C 180.000} C_DIS
LIN {X 125.970,Y 117.886,Z 54.049,A 180.000,B 0.000,C 180.000} C_DIS
LIN {X 125.984,Y 118.043,Z 54.046,A 180.000,B 0.000,C 180.000} C_DIS
LIN {X 125.989,Y 118.201,Z 54.043,A 180.000,B 0.000,C 180.000} C_DIS
LIN {X 125.994,Y 118.358,Z 54.040,A 180.000,B 0.000,C 180.000} C_DIS
LIN {X 125.998,Y 118.515,Z 54.037,A 180.000,B 0.000,C 180.000} C_DIS
LIN {X 125.993,Y 118.673,Z 54.034,A 180.000,B 0.000,C 180.000} C_DIS
LIN {X 125.988,Y 118.830,Z 54.032,A 180.000,B 0.000,C 180.000} C_DIS
LIN {X 125.982,Y 118.988,Z 54.029,A 180.000,B 0.000,C 180.000} C_DIS
LIN {X 125.968,Y 119.145,Z 54.027,A 180.000,B 0.000,C 180.000} C_DIS
LIN {X 125.937,Y 119.458,Z 54.022,A 180.000,B 0.000,C 180.000} C_DIS
LIN {X 125.887,Y 119.769,Z 54.018,A 180.000,B 0.000,C 180.000} C_DIS
LIN {X 125.827,Y 120.078,Z 54.014,A 180.000,B 0.000,C 180.000} C_DIS
LIN {X 125.757,Y 120.385,Z 54.011,A 180.000,B 0.000,C 180.000} C_DIS
LIN {X 125.669,Y 120.688,Z 54.008,A 180.000,B 0.000,C 180.000} C_DIS
LIN {X 125.571,Y 120.987,Z 54.005,A 180.000,B 0.000,C 180.000} C_DIS
LIN {X 125.463,Y 121.283,Z 54.003,A 180.000,B 0.000,C 180.000} C_DIS
LIN {X 125.337,Y 121.572,Z 54.002,A 180.000,B 0.000,C 180.000} C_DIS
LIN {X 125.202,Y 121.856,Z 54.001,A 180.000,B 0.000,C 180.000} C_DIS
LIN {X 125.057,Y 122.136,Z 54.000,A 180.000,B 0.000,C 180.000} C_DIS
LIN {X 124.939,Y 122.336,Z 54.000,A 180.000,B 0.000,C 180.000} C_DIS
; Cutting Move Starts
LIN {X 124.865,Y 122.461,Z 54.000,A 180.000,B 0.000,C 180.000} C_DIS
LIN {X 124.785,Y 122.587,Z 54.000,A 180.000,B 0.000,C 180.000} C_DIS
LIN {X 124.606,Y 122.850,Z 54.000,A 180.000,B 0.000,C 180.000} C_DIS
LIN {X 124.497,Y 122.997,Z 54.000,A 180.000,B 0.000,C 180.000} C_DIS
LIN {X 124.359,Y 123.176,Z 54.000,A 180.000,B 0.000,C 180.000} C_DIS
LIN {X 124.248,Y 123.313,Z 54.000,A 180.000,B 0.000,C 180.000} C_DIS
LIN {X 124.055,Y 123.533,Z 54.000,A 180.000,B 0.000,C 180.000} C_DIS
LIN {X 123.891,Y 123.709,Z 54.000,A 180.000,B 0.000,C 180.000} C_DIS
LIN {X 123.709,Y 123.891,Z 54.000,A 180.000,B 0.000,C 180.000} C_DIS
LIN {X 123.533,Y 124.055,Z 54.000,A 180.000,B 0.000,C 180.000} C_DIS
LIN {X 123.313,Y 124.248,Z 54.000,A 180.000,B 0.000,C 180.000} C_DIS
LIN {X 123.176,Y 124.359,Z 54.000,A 180.000,B 0.000,C 180.000} C_DIS
LIN {X 122.997,Y 124.497,Z 54.000,A 180.000,B 0.000,C 180.000} C_DIS
LIN {X 122.850,Y 124.606,Z 54.000,A 180.000,B 0.000,C 180.000} C_DIS
LIN {X 122.587,Y 124.785,Z 54.000,A 180.000,B 0.000,C 180.000} C_DIS
LIN {X 122.461,Y 124.865,Z 54.000,A 180.000,B 0.000,C 180.000} C_DIS
LIN {X 122.282,Y 124.971,Z 54.000,A 180.000,B 0.000,C 180.000} C_DIS
LIN {X 122.103,Y 125.076,Z 54.000,A 180.000,B 0.000,C 180.000} C_DIS
LIN {X 121.746,Y 125.258,Z 54.000,A 180.000,B 0.000,C 180.000} C_DIS
LIN {X 121.610,Y 125.321,Z 54.000,A 180.000,B 0.000,C 180.000} C_DIS
